LIN {X 0.009,Y -477.368,Z 1112.922,A 0.000,B 0.000,C 90.000,E1 22.025} C_DIS
LIN {X 0.039,Y -465.405,Z 1112.917,A 0.000,B 0.000,C 90.000,E1 20.972} C_DIS
LIN {X 0.095,Y -448.968,Z 1112.908,A 0.000,B 0.000,C 90.000,E1 19.504} C_DIS
LIN {X 0.026,Y -429.956,Z 1112.898,A 0.000,B 0.000,C 90.000,E1 17.692} C_DIS
LIN {X -0.246,Y -415.856,Z 1112.890,A 0.000,B 0.000,C 90.000,E1 16.205} C_DIS
LIN {X 0.123,Y -407.881,Z 1112.885,A 0.000,B 0.000,C 90.000,E1 15.190} C_DIS
LIN {X -0.086,Y -401.258,Z 1112.880,A 0.000,B 0.000,C 90.000,E1 14.356} C_DIS
LIN {X 0.152,Y -396.233,Z 1112.875,A 0.000,B 0.000,C 90.000,E1 13.536} C_DIS
LIN {X 0.076,Y -394.151,Z 1112.873,A 0.000,B 0.000,C 90.000,E1 13.119} C_DIS
LIN {X -0.071,Y -392.812,Z 1112.871,A 0.000,B 0.000,C 90.000,E1 12.703} C_DIS
LIN {X -0.136,Y -392.469,Z 1112.870,A 0.000,B 0.000,C 90.000,E1 12.535} C_DIS
LIN {X -0.161,Y -392.068,Z 1112.867,A 0.000,B 0.000,C 90.000,E1 12.007} C_DIS
LIN {X 0.211,Y -392.446,Z 1112.863,A 0.000,B 0.000,C 90.000,E1 11.243} C_DIS
LIN {X 0.042,Y -394.824,Z 1112.855,A 0.000,B 0.000,C 90.000,E1 9.849} C_DIS
LIN {X -0.112,Y -398.885,Z 1112.845,A 0.000,B 0.000,C 90.000,E1 8.106} C_DIS
LIN {X 0.165,Y -402.538,Z 1112.837,A 0.000,B 0.000,C 90.000,E1 6.663} C_DIS
LIN {X 0.148,Y -404.293,Z 1112.833,A 0.000,B 0.000,C 90.000,E1 5.967} C_DIS
LIN {X 0.101,Y -406.462,Z 1112.829,A 0.000,B 0.000,C 90.000,E1 5.277} C_DIS
LIN {X 0.083,Y -407.246,Z 1112.828,A 0.000,B 0.000,C 90.000,E1 5.106} C_DIS
LIN {X 0.015,Y -410.748,Z 1112.825,A 0.000,B 0.000,C 90.000,E1 4.531} C_DIS
LIN {X 0.005,Y -411.930,Z 1112.824,A 0.000,B 0.000,C 90.000,E1 4.359} C_DIS
LIN {X 0.157,Y -416.065,Z 1112.822,A 0.000,B 0.000,C 90.000,E1 3.955} C_DIS
LIN {X -0.197,Y -431.618,Z 1112.816,A 0.000,B 0.000,C 90.000,E1 2.922} C_DIS
LIN {X 0.226,Y -451.307,Z 1112.809,A 0.000,B 0.000,C 90.000,E1 1.547} C_DIS
LIN {X 0.037,Y -465.923,Z 1112.804,A 0.000,B 0.000,C 90.000,E1 0.630} C_DIS
LIN {X 0.181,Y -479.029,Z 1112.799,A 0.000,B 0.000,C 90.000,E1 359.771} C_DIS
LIN {X 0.170,Y -490.278,Z 1112.795,A 0.000,B 0.000,C 90.000,E1 359.026} C_DIS
LIN {X -0.165,Y -497.943,Z 1112.792,A 0.000,B 0.000,C 90.000,E1 358.511} C_DIS
LIN {X -0.165,Y -504.029,Z 1112.789,A 0.000,B 0.000,C 90.000,E1 358.051} C_DIS
LIN {X -0.251,Y -509.905,Z 1112.786,A 0.000,B 0.000,C 90.000,E1 357.593} C_DIS
LIN {X 0.073,Y -516.804,Z 1112.783,A 0.000,B 0.000,C 90.000,E1 356.963} C_DIS
LIN {X -0.071,Y -523.698,Z 1112.780,A 0.000,B 0.000,C 90.000,E1 356.331} C_DIS
LIN {X 0.049,Y -530.246,Z 1112.776,A 0.000,B 0.000,C 90.000,E1 355.641} C_DIS
LIN {X -0.178,Y -536.359,Z 1112.772,A 0.000,B 0.000,C 90.000,E1 354.951} C_DIS
LIN {X 0.132,Y -541.871,Z 1112.768,A 0.000,B 0.000,C 90.000,E1 354.204} C_DIS
LIN {X 0.212,Y -545.882,Z 1112.765,A 0.000,B 0.000,C 90.000,E1 353.628} C_DIS
LIN {X 0.129,Y -550.391,Z 1112.761,A 0.000,B 0.000,C 90.000,E1 352.932} C_DIS
LIN {X 0.274,Y -553.810,Z 1112.758,A 0.000,B 0.000,C 90.000,E1 352.356} C_DIS
LIN {X 0.269,Y -557.505,Z 1112.754,A 0.000,B 0.000,C 90.000,E1 351.659} C_DIS
LIN {X 0.210,Y -560.782,Z 1112.750,A 0.000,B 0.000,C 90.000,E1 350.971} C_DIS
LIN {X 0.112,Y -564.383,Z 1112.745,A 0.000,B 0.000,C 90.000,E1 350.151} C_DIS
LIN {X -0.050,Y -567.672,Z 1112.741,A 0.000,B 0.000,C 90.000,E1 349.342} C_DIS
LIN {X -0.075,Y -570.756,Z 1112.736,A 0.000,B 0.000,C 90.000,E1 348.522} C_DIS
LIN {X -0.065,Y -573.611,Z 1112.732,A 0.000,B 0.000,C 90.000,E1 347.701} C_DIS
LIN {X -0.025,Y -576.322,Z 1112.727,A 0.000,B 0.000,C 90.000,E1 346.881} C_DIS
LIN {X 0.039,Y -578.786,Z 1112.723,A 0.000,B 0.000,C 90.000,E1 346.061} C_DIS
LIN {X 0.154,Y -582.796,Z 1112.715,A 0.000,B 0.000,C 90.000,E1 344.700} C_DIS
LIN {X -0.131,Y -585.112,Z 1112.711,A 0.000,B 0.000,C 90.000,E1 343.921} C_DIS
LIN {X -0.065,Y -589.522,Z 1112.702,A 0.000,B 0.000,C 90.000,E1 342.308} C_DIS
LIN {X 0.024,Y -592.834,Z 1112.694,A 0.000,B 0.000,C 90.000,E1 340.967} C_DIS
LIN {X 0.287,Y -595.374,Z 1112.688,A 0.000,B 0.000,C 90.000,E1 339.880} C_DIS
LIN {X 0.329,Y -597.064,Z 1112.684,A 0.000,B 0.000,C 90.000,E1 339.082} C_DIS
LIN {X 0.079,Y -599.028,Z 1112.678,A 0.000,B 0.000,C 90.000,E1 338.050} C_DIS
LIN {X 0.070,Y -600.755,Z 1112.672,A 0.000,B 0.000,C 90.000,E1 336.997} C_DIS
LIN {X -0.154,Y -601.854,Z 1112.668,A 0.000,B 0.000,C 90.000,E1 336.230} C_DIS
LIN {X -0.127,Y -603.008,Z 1112.662,A 0.000,B 0.000,C 90.000,E1 335.177} C_DIS
LIN {X -0.319,Y -603.791,Z 1112.658,A 0.000,B 0.000,C 90.000,E1 334.409} C_DIS
LIN {X -0.019,Y -604.386,Z 1112.652,A 0.000,B 0.000,C 90.000,E1 333.332} C_DIS
LIN {X 0.081,Y -604.735,Z 1112.648,A 0.000,B 0.000,C 90.000,E1 332.538} C_DIS
LIN {X -0.208,Y -604.666,Z 1112.640,A 0.000,B 0.000,C 90.000,E1 331.257} C_DIS
LIN {X -0.156,Y -603.977,Z 1112.634,A 0.000,B 0.000,C 90.000,E1 330.205} C_DIS
LIN {X -0.049,Y -603.017,Z 1112.630,A 0.000,B 0.000,C 90.000,E1 329.410} C_DIS
LIN {X 0.121,Y -602.084,Z 1112.627,A 0.000,B 0.000,C 90.000,E1 328.869} C_DIS
LIN {X 0.206,Y -600.484,Z 1112.623,A 0.000,B 0.000,C 90.000,E1 328.074} C_DIS
LIN {X -0.235,Y -598.613,Z 1112.618,A 0.000,B 0.000,C 90.000,E1 327.327} C_DIS
LIN {X 0.132,Y -596.306,Z 1112.614,A 0.000,B 0.000,C 90.000,E1 326.501} C_DIS
LIN {X -0.016,Y -593.789,Z 1112.610,A 0.000,B 0.000,C 90.000,E1 325.722} C_DIS
LIN {X 0.300,Y -590.875,Z 1112.605,A 0.000,B 0.000,C 90.000,E1 324.895} C_DIS
LIN {X 0.103,Y -587.868,Z 1112.601,A 0.000,B 0.000,C 90.000,E1 324.116} C_DIS
LIN {X 0.154,Y -585.866,Z 1112.598,A 0.000,B 0.000,C 90.000,E1 323.577} C_DIS
LIN {X 0.067,Y -583.672,Z 1112.595,A 0.000,B 0.000,C 90.000,E1 323.050} C_DIS
LIN {X -0.032,Y -579.142,Z 1112.589,A 0.000,B 0.000,C 90.000,E1 321.984} C_DIS
LIN {X -0.155,Y -576.744,Z 1112.586,A 0.000,B 0.000,C 90.000,E1 321.457} C_DIS
LIN {X 0.044,Y -573.482,Z 1112.582,A 0.000,B 0.000,C 90.000,E1 320.759} C_DIS
LIN {X 0.067,Y -568.213,Z 1112.576,A 0.000,B 0.000,C 90.000,E1 319.666} C_DIS
LIN {X -0.255,Y -564.630,Z 1112.572,A 0.000,B 0.000,C 90.000,E1 319.013} C_DIS
LIN {X -0.102,Y -561.501,Z 1112.569,A 0.000,B 0.000,C 90.000,E1 318.447} C_DIS
LIN {X 0.074,Y -558.208,Z 1112.566,A 0.000,B 0.000,C 90.000,E1 317.877} C_DIS
LIN {X 0.183,Y -554.625,Z 1112.563,A 0.000,B 0.000,C 90.000,E1 317.310} C_DIS
LIN {X -0.049,Y -546.654,Z 1112.557,A 0.000,B 0.000,C 90.000,E1 316.215} C_DIS
LIN {X -0.215,Y -543.688,Z 1112.554,A 0.000,B 0.000,C 90.000,E1 315.810} C_DIS
LIN {X -0.008,Y -540.915,Z 1112.552,A 0.000,B 0.000,C 90.000,E1 315.364} C_DIS
LIN {X -0.214,Y -537.011,Z 1112.548,A 0.000,B 0.000,C 90.000,E1 314.676} C_DIS
LIN {X 0.330,Y -535.070,Z 1112.546,A 0.000,B 0.000,C 90.000,E1 314.190} C_DIS
LIN {X 0.005,Y -533.099,Z 1112.543,A 0.000,B 0.000,C 90.000,E1 313.662} C_DIS
LIN {X 0.029,Y -531.114,Z 1112.538,A 0.000,B 0.000,C 90.000,E1 312.894} C_DIS
LIN {X 0.003,Y -530.609,Z 1112.537,A 0.000,B 0.000,C 90.000,E1 312.609} C_DIS
LIN {X -0.084,Y -529.964,Z 1112.534,A 0.000,B 0.000,C 90.000,E1 312.043} C_DIS
LIN {X -0.111,Y -529.478,Z 1112.532,A 0.000,B 0.000,C 90.000,E1 311.757} C_DIS
LIN {X -0.136,Y -529.401,Z 1112.530,A 0.000,B 0.000,C 90.000,E1 311.472} C_DIS
LIN {X 0.162,Y -528.898,Z 1112.527,A 0.000,B 0.000,C 90.000,E1 310.862} C_DIS
LIN {X 0.052,Y -528.782,Z 1112.524,A 0.000,B 0.000,C 90.000,E1 310.297} C_DIS
LIN {X 0.290,Y -528.759,Z 1112.518,A 0.000,B 0.000,C 90.000,E1 309.116} C_DIS
LIN {X 0.096,Y -529.954,Z 1112.501,A 0.000,B 0.000,C 90.000,E1 306.251} C_DIS
LIN {X -0.018,Y -531.286,Z 1112.490,A 0.000,B 0.000,C 90.000,E1 304.246} C_DIS
LIN {X -0.260,Y -532.419,Z 1112.481,A 0.000,B 0.000,C 90.000,E1 302.546} C_DIS
LIN {X -0.019,Y -533.825,Z 1112.471,A 0.000,B 0.000,C 90.000,E1 300.797} C_DIS
LIN {X -0.020,Y -535.088,Z 1112.462,A 0.000,B 0.000,C 90.000,E1 299.077} C_DIS
LIN {X -0.141,Y -535.607,Z 1112.457,A 0.000,B 0.000,C 90.000,E1 298.231} C_DIS
LIN {X -0.092,Y -536.415,Z 1112.449,A 0.000,B 0.000,C 90.000,E1 296.796} C_DIS
LIN {X 0.038,Y -536.763,Z 1112.444,A 0.000,B 0.000,C 90.000,E1 295.924} C_DIS
LIN {X -0.139,Y -537.151,Z 1112.436,A 0.000,B 0.000,C 90.000,E1 294.515} C_DIS
LIN {X -0.051,Y -537.438,Z 1112.428,A 0.000,B 0.000,C 90.000,E1 293.078} C_DIS
LIN {X -0.161,Y -537.544,Z 1112.420,A 0.000,B 0.000,C 90.000,E1 291.663} C_DIS
LIN {X -0.266,Y -537.534,Z 1112.412,A 0.000,B 0.000,C 90.000,E1 290.248} C_DIS
LIN {X -0.089,Y -537.427,Z 1112.406,A 0.000,B 0.000,C 90.000,E1 289.087} C_DIS
LIN {X -0.139,Y -536.979,Z 1112.395,A 0.000,B 0.000,C 90.000,E1 287.094} C_DIS
LIN {X -0.046,Y -536.434,Z 1112.385,A 0.000,B 0.000,C 90.000,E1 285.371} C_DIS
LIN {X -0.207,Y -535.915,Z 1112.379,A 0.000,B 0.000,C 90.000,E1 284.245} C_DIS
LIN {X -0.214,Y -534.929,Z 1112.368,A 0.000,B 0.000,C 90.000,E1 282.243} C_DIS
LIN {X 0.058,Y -534.206,Z 1112.360,A 0.000,B 0.000,C 90.000,E1 280.782} C_DIS
LIN {X -0.170,Y -533.353,Z 1112.350,A 0.000,B 0.000,C 90.000,E1 279.086} C_DIS
LIN {X -0.096,Y -532.371,Z 1112.339,A 0.000,B 0.000,C 90.000,E1 277.068} C_DIS
LIN {X -0.039,Y -531.638,Z 1112.331,A 0.000,B 0.000,C 90.000,E1 275.625} C_DIS
LIN {X -0.051,Y -530.744,Z 1112.320,A 0.000,B 0.000,C 90.000,E1 273.612} C_DIS
LIN {X -0.111,Y -530.074,Z 1112.312,A 0.000,B 0.000,C 90.000,E1 272.178} C_DIS
LIN {X -0.203,Y -529.294,Z 1112.302,A 0.000,B 0.000,C 90.000,E1 270.458} C_DIS
LIN {X -0.262,Y -528.907,Z 1112.298,A 0.000,B 0.000,C 90.000,E1 269.599} C_DIS
LIN {X 0.149,Y -528.050,Z 1112.288,A 0.000,B 0.000,C 90.000,E1 267.822} C_DIS
LIN {X 0.038,Y -527.174,Z 1112.280,A 0.000,B 0.000,C 90.000,E1 266.388} C_DIS
LIN {X -0.096,Y -526.057,Z 1112.270,A 0.000,B 0.000,C 90.000,E1 264.666} C_DIS
LIN {X -0.173,Y -525.177,Z 1112.264,A 0.000,B 0.000,C 90.000,E1 263.514} C_DIS
LIN {X -0.197,Y -524.077,Z 1112.257,A 0.000,B 0.000,C 90.000,E1 262.356} C_DIS
LIN {X 0.232,Y -521.513,Z 1112.243,A 0.000,B 0.000,C 90.000,E1 259.690} C_DIS
LIN {X 0.247,Y -519.858,Z 1112.233,A 0.000,B 0.000,C 90.000,E1 257.937} C_DIS
LIN {X -0.175,Y -517.933,Z 1112.222,A 0.000,B 0.000,C 90.000,E1 255.936} C_DIS
LIN {X -0.100,Y -516.792,Z 1112.215,A 0.000,B 0.000,C 90.000,E1 254.755} C_DIS
LIN {X 0.095,Y -515.517,Z 1112.209,A 0.000,B 0.000,C 90.000,E1 253.559} C_DIS
LIN {X -0.136,Y -513.723,Z 1112.199,A 0.000,B 0.000,C 90.000,E1 251.819} C_DIS
LIN {X 0.120,Y -512.149,Z 1112.191,A 0.000,B 0.000,C 90.000,E1 250.315} C_DIS
LIN {X 0.139,Y -510.097,Z 1112.181,A 0.000,B 0.000,C 90.000,E1 248.539} C_DIS
LIN {X -0.166,Y -507.911,Z 1112.171,A 0.000,B 0.000,C 90.000,E1 246.794} C_DIS
LIN {X 0.129,Y -506.655,Z 1112.166,A 0.000,B 0.000,C 90.000,E1 245.869} C_DIS
LIN {X -0.216,Y -504.978,Z 1112.159,A 0.000,B 0.000,C 90.000,E1 244.717} C_DIS
LIN {X -0.124,Y -503.108,Z 1112.153,A 0.000,B 0.000,C 90.000,E1 243.512} C_DIS
LIN {X 0.077,Y -500.227,Z 1112.143,A 0.000,B 0.000,C 90.000,E1 241.691} C_DIS
LIN {X 0.031,Y -498.747,Z 1112.138,A 0.000,B 0.000,C 90.000,E1 240.795} C_DIS
LIN {X -0.059,Y -495.801,Z 1112.128,A 0.000,B 0.000,C 90.000,E1 238.997} C_DIS
LIN {X -0.069,Y -493.686,Z 1112.121,A 0.000,B 0.000,C 90.000,E1 237.788} C_DIS
LIN {X -0.020,Y -490.521,Z 1112.111,A 0.000,B 0.000,C 90.000,E1 235.960} C_DIS
LIN {X 0.264,Y -487.817,Z 1112.102,A 0.000,B 0.000,C 90.000,E1 234.402} C_DIS
LIN {X -0.179,Y -484.923,Z 1112.094,A 0.000,B 0.000,C 90.000,E1 232.924} C_DIS
LIN {X 0.104,Y -481.406,Z 1112.084,A 0.000,B 0.000,C 90.000,E1 231.045} C_DIS
LIN {X -0.048,Y -479.034,Z 1112.077,A 0.000,B 0.000,C 90.000,E1 229.828} C_DIS
LIN {X 0.237,Y -476.005,Z 1112.068,A 0.000,B 0.000,C 90.000,E1 228.243} C_DIS
LIN {X 0.200,Y -472.520,Z 1112.058,A 0.000,B 0.000,C 90.000,E1 226.377} C_DIS
LIN {X 0.070,Y -469.061,Z 1112.047,A 0.000,B 0.000,C 90.000,E1 224.514} C_DIS
LIN {X 0.130,Y -466.300,Z 1112.039,A 0.000,B 0.000,C 90.000,E1 222.933} C_DIS
LIN {X -0.121,Y -463.116,Z 1112.028,A 0.000,B 0.000,C 90.000,E1 221.067} C_DIS
LIN {X -0.012,Y -459.634,Z 1112.016,A 0.000,B 0.000,C 90.000,E1 218.830} C_DIS
LIN {X 0.075,Y -456.279,Z 1112.003,A 0.000,B 0.000,C 90.000,E1 216.583} C_DIS
LIN {X 0.090,Y -454.065,Z 1111.994,A 0.000,B 0.000,C 90.000,E1 214.978} C_DIS
LIN {X 0.063,Y -451.814,Z 1111.985,A 0.000,B 0.000,C 90.000,E1 213.372} C_DIS
LIN {X -0.099,Y -448.884,Z 1111.973,A 0.000,B 0.000,C 90.000,E1 211.131} C_DIS
LIN {X 0.198,Y -446.213,Z 1111.960,A 0.000,B 0.000,C 90.000,E1 208.821} C_DIS
LIN {X 0.006,Y -444.131,Z 1111.948,A 0.000,B 0.000,C 90.000,E1 206.565} C_DIS
LIN {X 0.114,Y -443.057,Z 1111.937,A 0.000,B 0.000,C 90.000,E1 204.591} C_DIS
LIN {X 0.156,Y -443.425,Z 1111.928,A 0.000,B 0.000,C 90.000,E1 202.950} C_DIS
LIN {X 0.002,Y -444.595,Z 1111.920,A 0.000,B 0.000,C 90.000,E1 201.663} C_DIS
LIN {X -0.114,Y -445.583,Z 1111.917,A 0.000,B 0.000,C 90.000,E1 201.025} C_DIS
LIN {X -0.259,Y -447.580,Z 1111.911,A 0.000,B 0.000,C 90.000,E1 200.066} C_DIS
LIN {X -0.044,Y -451.809,Z 1111.902,A 0.000,B 0.000,C 90.000,E1 198.417} C_DIS
LIN {X 0.073,Y -459.189,Z 1111.890,A 0.000,B 0.000,C 90.000,E1 196.150} C_DIS
LIN {X 0.227,Y -470.714,Z 1111.873,A 0.000,B 0.000,C 90.000,E1 193.119} C_DIS
LIN {X 0.094,Y -479.895,Z 1111.861,A 0.000,B 0.000,C 90.000,E1 190.950} C_DIS
LIN {X -0.116,Y -488.663,Z 1111.850,A 0.000,B 0.000,C 90.000,E1 188.973} C_DIS
LIN {X -0.095,Y -496.045,Z 1111.841,A 0.000,B 0.000,C 90.000,E1 187.296} C_DIS
LIN {X -0.165,Y -502.571,Z 1111.832,A 0.000,B 0.000,C 90.000,E1 185.796} C_DIS
LIN {X 0.188,Y -511.586,Z 1111.821,A 0.000,B 0.000,C 90.000,E1 183.669} C_DIS
LIN {X 0.112,Y -517.370,Z 1111.813,A 0.000,B 0.000,C 90.000,E1 182.350} C_DIS
LIN {X 0.047,Y -525.847,Z 1111.803,A 0.000,B 0.000,C 90.000,E1 180.458} C_DIS
LIN {X 0.182,Y -532.968,Z 1111.794,A 0.000,B 0.000,C 90.000,E1 178.854} C_DIS
LIN {X -0.065,Y -540.073,Z 1111.785,A 0.000,B 0.000,C 90.000,E1 177.306} C_DIS
LIN {X 0.112,Y -546.498,Z 1111.777,A 0.000,B 0.000,C 90.000,E1 175.869} C_DIS
LIN {X 0.064,Y -552.222,Z 1111.770,A 0.000,B 0.000,C 90.000,E1 174.609} C_DIS
LIN {X -0.145,Y -560.503,Z 1111.760,A 0.000,B 0.000,C 90.000,E1 172.818} C_DIS
LIN {X -0.095,Y -566.810,Z 1111.752,A 0.000,B 0.000,C 90.000,E1 171.432} C_DIS
LIN {X -0.085,Y -573.537,Z 1111.744,A 0.000,B 0.000,C 90.000,E1 169.926} C_DIS
LIN {X -0.182,Y -579.558,Z 1111.736,A 0.000,B 0.000,C 90.000,E1 168.578} C_DIS
LIN {X 0.158,Y -584.140,Z 1111.730,A 0.000,B 0.000,C 90.000,E1 167.465} C_DIS
LIN {X -0.259,Y -587.510,Z 1111.726,A 0.000,B 0.000,C 90.000,E1 166.700} C_DIS
LIN {X 0.184,Y -591.788,Z 1111.720,A 0.000,B 0.000,C 90.000,E1 165.589} C_DIS
LIN {X -0.013,Y -594.883,Z 1111.716,A 0.000,B 0.000,C 90.000,E1 164.810} C_DIS
LIN {X -0.183,Y -599.654,Z 1111.708,A 0.000,B 0.000,C 90.000,E1 163.504} C_DIS
LIN {X -0.296,Y -602.396,Z 1111.704,A 0.000,B 0.000,C 90.000,E1 162.725} C_DIS
LIN {X -0.170,Y -606.635,Z 1111.697,A 0.000,B 0.000,C 90.000,E1 161.402} C_DIS
LIN {X -0.286,Y -609.858,Z 1111.691,A 0.000,B 0.000,C 90.000,E1 160.369} C_DIS
LIN {X -0.144,Y -612.911,Z 1111.685,A 0.000,B 0.000,C 90.000,E1 159.316} C_DIS
LIN {X -0.174,Y -615.788,Z 1111.679,A 0.000,B 0.000,C 90.000,E1 158.284} C_DIS
LIN {X -0.219,Y -619.981,Z 1111.671,A 0.000,B 0.000,C 90.000,E1 156.741} C_DIS
LIN {X 0.057,Y -623.295,Z 1111.664,A 0.000,B 0.000,C 90.000,E1 155.433} C_DIS
LIN {X 0.076,Y -625.894,Z 1111.658,A 0.000,B 0.000,C 90.000,E1 154.409} C_DIS
LIN {X 0.157,Y -628.951,Z 1111.651,A 0.000,B 0.000,C 90.000,E1 153.127} C_DIS
LIN {X -0.271,Y -631.792,Z 1111.644,A 0.000,B 0.000,C 90.000,E1 151.897} C_DIS
LIN {X 0.205,Y -634.592,Z 1111.637,A 0.000,B 0.000,C 90.000,E1 150.589} C_DIS
LIN {X 0.220,Y -637.771,Z 1111.628,A 0.000,B 0.000,C 90.000,E1 149.076} C_DIS
LIN {X -0.309,Y -640.299,Z 1111.621,A 0.000,B 0.000,C 90.000,E1 147.867} C_DIS
LIN {X 0.081,Y -642.717,Z 1111.614,A 0.000,B 0.000,C 90.000,E1 146.580} C_DIS
LIN {X -0.076,Y -644.570,Z 1111.609,A 0.000,B 0.000,C 90.000,E1 145.595} C_DIS
LIN {X -0.156,Y -646.753,Z 1111.602,A 0.000,B 0.000,C 90.000,E1 144.356} C_DIS
LIN {X 0.084,Y -649.389,Z 1111.594,A 0.000,B 0.000,C 90.000,E1 142.844} C_DIS
LIN {X -0.156,Y -652.964,Z 1111.583,A 0.000,B 0.000,C 90.000,E1 140.884} C_DIS
LIN {X -0.400,Y -656.643,Z 1111.572,A 0.000,B 0.000,C 90.000,E1 138.933} C_DIS
LIN {X 0.354,Y -660.001,Z 1111.562,A 0.000,B 0.000,C 90.000,E1 137.148} C_DIS
LIN {X -0.236,Y -664.132,Z 1111.551,A 0.000,B 0.000,C 90.000,E1 135.243} C_DIS
LIN {X 0.230,Y -669.230,Z 1111.539,A 0.000,B 0.000,C 90.000,E1 133.014} C_DIS
LIN {X -0.060,Y -674.540,Z 1111.527,A 0.000,B 0.000,C 90.000,E1 130.862} C_DIS
LIN {X 0.138,Y -678.079,Z 1111.519,A 0.000,B 0.000,C 90.000,E1 129.402} C_DIS
LIN {X 0.070,Y -681.801,Z 1111.511,A 0.000,B 0.000,C 90.000,E1 127.971} C_DIS
LIN {X 0.088,Y -685.476,Z 1111.503,A 0.000,B 0.000,C 90.000,E1 126.537} C_DIS
LIN {X 0.325,Y -687.268,Z 1111.499,A 0.000,B 0.000,C 90.000,E1 125.804} C_DIS
LIN {X -0.325,Y -691.332,Z 1111.490,A 0.000,B 0.000,C 90.000,E1 124.199} C_DIS
LIN {X 0.036,Y -694.817,Z 1111.482,A 0.000,B 0.000,C 90.000,E1 122.752} C_DIS
LIN {X 0.185,Y -697.012,Z 1111.477,A 0.000,B 0.000,C 90.000,E1 121.799} C_DIS
LIN {X -0.257,Y -698.517,Z 1111.473,A 0.000,B 0.000,C 90.000,E1 121.131} C_DIS
LIN {X -0.082,Y -699.870,Z 1111.469,A 0.000,B 0.000,C 90.000,E1 120.413} C_DIS
LIN {X 0.119,Y -701.498,Z 1111.464,A 0.000,B 0.000,C 90.000,E1 119.461} C_DIS
LIN {X -0.015,Y -702.954,Z 1111.459,A 0.000,B 0.000,C 90.000,E1 118.537} C_DIS
LIN {X 0.158,Y -704.253,Z 1111.453,A 0.000,B 0.000,C 90.000,E1 117.590} C_DIS
LIN {X -0.236,Y -704.918,Z 1111.449,A 0.000,B 0.000,C 90.000,E1 116.924} C_DIS
LIN {X 0.262,Y -705.762,Z 1111.443,A 0.000,B 0.000,C 90.000,E1 115.720} C_DIS
LIN {X 0.195,Y -705.963,Z 1111.439,A 0.000,B 0.000,C 90.000,E1 115.027} C_DIS
LIN {X -0.158,Y -705.902,Z 1111.437,A 0.000,B 0.000,C 90.000,E1 114.591} C_DIS
LIN {X -0.221,Y -705.136,Z 1111.434,A 0.000,B 0.000,C 90.000,E1 114.131} C_DIS
LIN {X -0.220,Y -704.594,Z 1111.433,A 0.000,B 0.000,C 90.000,E1 113.898} C_DIS
LIN {X 0.348,Y -702.685,Z 1111.430,A 0.000,B 0.000,C 90.000,E1 113.387} C_DIS
LIN {X -0.436,Y -702.113,Z 1111.429,A 0.000,B 0.000,C 90.000,E1 113.334} C_DIS
LIN {X -0.297,Y -701.240,Z 1111.429,A 0.000,B 0.000,C 90.000,E1 113.206} C_DIS
LIN {X -0.029,Y -696.964,Z 1111.426,A 0.000,B 0.000,C 90.000,E1 112.717} C_DIS
LIN {X 0.099,Y -695.384,Z 1111.426,A 0.000,B 0.000,C 90.000,E1 112.589} C_DIS
LIN {X -0.014,Y -690.978,Z 1111.425,A 0.000,B 0.000,C 90.000,E1 112.408} C_DIS
LIN {X -0.072,Y -685.718,Z 1111.423,A 0.000,B 0.000,C 90.000,E1 112.206} C_DIS
LIN {X 0.066,Y -683.449,Z 1111.423,A 0.000,B 0.000,C 90.000,E1 112.153} C_DIS
LIN {X 0.059,Y -676.047,Z 1111.423,A 0.000,B 0.000,C 90.000,E1 112.078} C_DIS
LIN {X 0.013,Y -603.763,Z 1111.423,A 0.000,B 0.000,C 90.000,E1 112.078} C_DIS
LIN {X 0.029,Y -600.557,Z 1111.422,A 0.000,B 0.000,C 90.000,E1 111.897} C_DIS
LIN {X 0.111,Y -594.792,Z 1111.419,A 0.000,B 0.000,C 90.000,E1 111.461} C_DIS
LIN {X 0.166,Y -587.133,Z 1111.416,A 0.000,B 0.000,C 90.000,E1 110.791} C_DIS
LIN {X 0.151,Y -578.854,Z 1111.412,A 0.000,B 0.000,C 90.000,E1 110.066} C_DIS
LIN {X 0.192,Y -574.638,Z 1111.410,A 0.000,B 0.000,C 90.000,E1 109.704} C_DIS
LIN {X -0.003,Y -568.549,Z 1111.407,A 0.000,B 0.000,C 90.000,E1 109.268} C_DIS
LIN {X 0.255,Y -560.311,Z 1111.404,A 0.000,B 0.000,C 90.000,E1 108.725} C_DIS
LIN {X 0.085,Y -553.963,Z 1111.402,A 0.000,B 0.000,C 90.000,E1 108.362} C_DIS
LIN {X -0.188,Y -550.006,Z 1111.401,A 0.000,B 0.000,C 90.000,E1 108.109} C_DIS
LIN {X 0.258,Y -548.776,Z 1111.400,A 0.000,B 0.000,C 90.000,E1 107.873} C_DIS
LIN {X 0.216,Y -548.757,Z 1111.399,A 0.000,B 0.000,C 90.000,E1 107.873} C_DIS
LIN {X -0.099,Y -548.411,Z 1111.397,A 0.000,B 0.000,C 90.000,E1 107.511} C_DIS
LIN {X 0.075,Y -548.753,Z 1111.393,A 0.000,B 0.000,C 90.000,E1 106.732} C_DIS
LIN {X 0.084,Y -549.554,Z 1111.387,A 0.000,B 0.000,C 90.000,E1 105.607} C_DIS
LIN {X 0.261,Y -551.471,Z 1111.373,A 0.000,B 0.000,C 90.000,E1 103.063} C_DIS
LIN {X 0.009,Y -553.177,Z 1111.362,A 0.000,B 0.000,C 90.000,E1 101.130} C_DIS
LIN {X 0.114,Y -554.811,Z 1111.353,A 0.000,B 0.000,C 90.000,E1 99.443} C_DIS
LIN {X 0.250,Y -556.528,Z 1111.343,A 0.000,B 0.000,C 90.000,E1 97.757} C_DIS
LIN {X -0.158,Y -558.492,Z 1111.333,A 0.000,B 0.000,C 90.000,E1 95.853} C_DIS
LIN {X -0.230,Y -559.689,Z 1111.325,A 0.000,B 0.000,C 90.000,E1 94.473} C_DIS
LIN {X 0.274,Y -560.766,Z 1111.317,A 0.000,B 0.000,C 90.000,E1 93.037} C_DIS
LIN {X 0.089,Y -561.446,Z 1111.311,A 0.000,B 0.000,C 90.000,E1 91.949} C_DIS
LIN {X 0.035,Y -562.276,Z 1111.303,A 0.000,B 0.000,C 90.000,E1 90.573} C_DIS
LIN {X -0.018,Y -562.972,Z 1111.296,A 0.000,B 0.000,C 90.000,E1 89.198} C_DIS
LIN {X 0.058,Y -563.839,Z 1111.286,A 0.000,B 0.000,C 90.000,E1 87.535} C_DIS
LIN {X 0.185,Y -564.611,Z 1111.277,A 0.000,B 0.000,C 90.000,E1 85.869} C_DIS
LIN {X -0.082,Y -565.364,Z 1111.266,A 0.000,B 0.000,C 90.000,E1 83.970} C_DIS
LIN {X 0.290,Y -566.130,Z 1111.256,A 0.000,B 0.000,C 90.000,E1 82.008} C_DIS
LIN {X 0.191,Y -566.832,Z 1111.245,A 0.000,B 0.000,C 90.000,E1 80.095} C_DIS
LIN {X 0.022,Y -567.505,Z 1111.236,A 0.000,B 0.000,C 90.000,E1 78.465} C_DIS
LIN {X -0.026,Y -568.295,Z 1111.227,A 0.000,B 0.000,C 90.000,E1 76.825} C_DIS
LIN {X 0.199,Y -569.676,Z 1111.213,A 0.000,B 0.000,C 90.000,E1 74.338} C_DIS
LIN {X -0.097,Y -571.244,Z 1111.201,A 0.000,B 0.000,C 90.000,E1 72.181} C_DIS
LIN {X 0.182,Y -573.217,Z 1111.187,A 0.000,B 0.000,C 90.000,E1 69.699} C_DIS
LIN {X 0.192,Y -574.425,Z 1111.180,A 0.000,B 0.000,C 90.000,E1 68.337} C_DIS
LIN {X 0.231,Y -575.716,Z 1111.172,A 0.000,B 0.000,C 90.000,E1 66.975} C_DIS
LIN {X -0.018,Y -577.324,Z 1111.162,A 0.000,B 0.000,C 90.000,E1 65.101} C_DIS
LIN {X -0.230,Y -578.399,Z 1111.154,A 0.000,B 0.000,C 90.000,E1 63.768} C_DIS
LIN {X 0.208,Y -579.564,Z 1111.145,A 0.000,B 0.000,C 90.000,E1 62.103} C_DIS
LIN {X -0.216,Y -580.819,Z 1111.135,A 0.000,B 0.000,C 90.000,E1 60.255} C_DIS
LIN {X 0.172,Y -581.619,Z 1111.127,A 0.000,B 0.000,C 90.000,E1 58.869} C_DIS
LIN {X 0.212,Y -582.297,Z 1111.121,A 0.000,B 0.000,C 90.000,E1 57.788} C_DIS
LIN {X -0.026,Y -583.232,Z 1111.111,A 0.000,B 0.000,C 90.000,E1 55.928} C_DIS
LIN {X -0.090,Y -584.056,Z 1111.102,A 0.000,B 0.000,C 90.000,E1 54.322} C_DIS
LIN {X -0.245,Y -584.944,Z 1111.090,A 0.000,B 0.000,C 90.000,E1 52.190} C_DIS
LIN {X 0.040,Y -585.158,Z 1111.084,A 0.000,B 0.000,C 90.000,E1 51.090} C_DIS
LIN {X 0.144,Y -585.281,Z 1111.079,A 0.000,B 0.000,C 90.000,E1 50.275} C_DIS
LIN {X 0.165,Y -585.200,Z 1111.072,A 0.000,B 0.000,C 90.000,E1 48.933} C_DIS
LIN {X -0.002,Y -585.032,Z 1111.066,A 0.000,B 0.000,C 90.000,E1 47.877} C_DIS
LIN {X 0.218,Y -584.729,Z 1111.060,A 0.000,B 0.000,C 90.000,E1 46.782} C_DIS
LIN {X -0.245,Y -584.197,Z 1111.053,A 0.000,B 0.000,C 90.000,E1 45.486} C_DIS
LIN {X -0.044,Y -583.562,Z 1111.047,A 0.000,B 0.000,C 90.000,E1 44.393} C_DIS
LIN {X 0.012,Y -582.954,Z 1111.042,A 0.000,B 0.000,C 90.000,E1 43.581} C_DIS
LIN {X -0.217,Y -581.967,Z 1111.036,A 0.000,B 0.000,C 90.000,E1 42.528} C_DIS
LIN {X 0.068,Y -581.311,Z 1111.033,A 0.000,B 0.000,C 90.000,E1 41.962} C_DIS
LIN {X -0.156,Y -579.979,Z 1111.027,A 0.000,B 0.000,C 90.000,E1 40.906} C_DIS
LIN {X -0.112,Y -578.921,Z 1111.023,A 0.000,B 0.000,C 90.000,E1 40.092} C_DIS
LIN {X -0.208,Y -576.639,Z 1111.015,A 0.000,B 0.000,C 90.000,E1 38.749} C_DIS
LIN {X 0.254,Y -575.062,Z 1111.011,A 0.000,B 0.000,C 90.000,E1 37.890} C_DIS
LIN {X 0.245,Y -573.236,Z 1111.006,A 0.000,B 0.000,C 90.000,E1 37.076} C_DIS
LIN {X -0.129,Y -571.225,Z 1111.002,A 0.000,B 0.000,C 90.000,E1 36.297} C_DIS
LIN {X 0.008,Y -570.520,Z 1111.000,A 0.000,B 0.000,C 90.000,E1 36.011} C_DIS
LIN {X 0.070,Y -567.941,Z 1110.996,A 0.000,B 0.000,C 90.000,E1 35.185} C_DIS
LIN {X -0.354,Y -565.171,Z 1110.991,A 0.000,B 0.000,C 90.000,E1 34.405} C_DIS
LIN {X -0.242,Y -564.159,Z 1110.990,A 0.000,B 0.000,C 90.000,E1 34.119} C_DIS
LIN {X -0.242,Y -560.733,Z 1110.985,A 0.000,B 0.000,C 90.000,E1 33.293} C_DIS
LIN {X 0.191,Y -557.057,Z 1110.980,A 0.000,B 0.000,C 90.000,E1 32.418} C_DIS
LIN {X 0.104,Y -552.952,Z 1110.976,A 0.000,B 0.000,C 90.000,E1 31.592} C_DIS
LIN {X -0.196,Y -549.302,Z 1110.972,A 0.000,B 0.000,C 90.000,E1 30.924} C_DIS
LIN {X -0.176,Y -544.633,Z 1110.967,A 0.000,B 0.000,C 90.000,E1 30.079} C_DIS
LIN {X 0.196,Y -540.523,Z 1110.963,A 0.000,B 0.000,C 90.000,E1 29.333} C_DIS
LIN {X -0.335,Y -536.954,Z 1110.960,A 0.000,B 0.000,C 90.000,E1 28.821} C_DIS
LIN {X -0.158,Y -533.062,Z 1110.957,A 0.000,B 0.000,C 90.000,E1 28.231} C_DIS
LIN {X -0.161,Y -527.800,Z 1110.953,A 0.000,B 0.000,C 90.000,E1 27.513} C_DIS
LIN {X -0.058,Y -523.395,Z 1110.950,A 0.000,B 0.000,C 90.000,E1 26.924} C_DIS
LIN {X -0.062,Y -519.909,Z 1110.947,A 0.000,B 0.000,C 90.000,E1 26.488} C_DIS
LIN {X 0.292,Y -513.604,Z 1110.943,A 0.000,B 0.000,C 90.000,E1 25.720} C_DIS
LIN {X -0.129,Y -505.696,Z 1110.938,A 0.000,B 0.000,C 90.000,E1 24.899} C_DIS
LIN {X -0.083,Y -496.065,Z 1110.933,A 0.000,B 0.000,C 90.000,E1 23.898} C_DIS
LIN {X -0.165,Y -486.110,Z 1110.927,A 0.000,B 0.000,C 90.000,E1 22.950} C_DIS
LIN {X -0.178,Y -477.456,Z 1110.923,A 0.000,B 0.000,C 90.000,E1 22.153} C_DIS
LIN {X 0.185,Y -470.038,Z 1110.919,A 0.000,B 0.000,C 90.000,E1 21.461} C_DIS
LIN {X -0.138,Y -457.051,Z 1110.913,A 0.000,B 0.000,C 90.000,E1 20.355} C_DIS
LIN {X 0.015,Y -435.079,Z 1110.902,A 0.000,B 0.000,C 90.000,E1 18.308} C_DIS
LIN {X 0.093,Y -422.326,Z 1110.895,A 0.000,B 0.000,C 90.000,E1 16.985} C_DIS
LIN {X -0.219,Y -411.437,Z 1110.888,A 0.000,B 0.000,C 90.000,E1 15.788} C_DIS
LIN {X 0.025,Y -401.084,Z 1110.880,A 0.000,B 0.000,C 90.000,E1 14.426} C_DIS
LIN {X 0.078,Y -396.147,Z 1110.876,A 0.000,B 0.000,C 90.000,E1 13.647} C_DIS
LIN {X 0.048,Y -394.506,Z 1110.874,A 0.000,B 0.000,C 90.000,E1 13.300} C_DIS
LIN {X 0.074,Y -393.770,Z 1110.873,A 0.000,B 0.000,C 90.000,E1 13.119} C_DIS
LIN {X -0.137,Y -392.324,Z 1110.870,A 0.000,B 0.000,C 90.000,E1 12.591} C_DIS
LIN {X 0.138,Y -391.973,Z 1110.867,A 0.000,B 0.000,C 90.000,E1 12.007} C_DIS
LIN {X -0.119,Y -392.534,Z 1110.863,A 0.000,B 0.000,C 90.000,E1 11.299} C_DIS
LIN {X 0.063,Y -395.659,Z 1110.853,A 0.000,B 0.000,C 90.000,E1 9.500} C_DIS
LIN {X -0.053,Y -398.954,Z 1110.845,A 0.000,B 0.000,C 90.000,E1 8.106} C_DIS
LIN {X -0.173,Y -402.562,Z 1110.837,A 0.000,B 0.000,C 90.000,E1 6.720} C_DIS
LIN {X 0.210,Y -404.272,Z 1110.833,A 0.000,B 0.000,C 90.000,E1 5.967} C_DIS
LIN {X 0.163,Y -406.373,Z 1110.829,A 0.000,B 0.000,C 90.000,E1 5.277} C_DIS
LIN {X 0.146,Y -407.055,Z 1110.828,A 0.000,B 0.000,C 90.000,E1 5.106} C_DIS
LIN {X -0.132,Y -410.515,Z 1110.825,A 0.000,B 0.000,C 90.000,E1 4.531} C_DIS
LIN {X -0.144,Y -411.729,Z 1110.824,A 0.000,B 0.000,C 90.000,E1 4.359} C_DIS
LIN {X 0.000,Y -415.683,Z 1110.822,A 0.000,B 0.000,C 90.000,E1 3.955} C_DIS
LIN {X 0.208,Y -417.440,Z 1110.821,A 0.000,B 0.000,C 90.000,E1 3.784} C_DIS
LIN {X -0.031,Y -426.335,Z 1110.818,A 0.000,B 0.000,C 90.000,E1 3.212} C_DIS
LIN {X -0.183,Y -446.085,Z 1110.810,A 0.000,B 0.000,C 90.000,E1 1.892} C_DIS
LIN {X -0.185,Y -465.636,Z 1110.803,A 0.000,B 0.000,C 90.000,E1 0.630} C_DIS
LIN {X 0.181,Y -478.333,Z 1110.799,A 0.000,B 0.000,C 90.000,E1 359.771} C_DIS
LIN {X 0.122,Y -488.018,Z 1110.795,A 0.000,B 0.000,C 90.000,E1 359.141} C_DIS
LIN {X -0.161,Y -495.830,Z 1110.792,A 0.000,B 0.000,C 90.000,E1 358.625} C_DIS
LIN {X -0.118,Y -503.463,Z 1110.789,A 0.000,B 0.000,C 90.000,E1 358.051} C_DIS
LIN {X -0.235,Y -509.453,Z 1110.786,A 0.000,B 0.000,C 90.000,E1 357.593} C_DIS
LIN {X -0.022,Y -516.607,Z 1110.783,A 0.000,B 0.000,C 90.000,E1 356.963} C_DIS
LIN {X -0.148,Y -523.521,Z 1110.780,A 0.000,B 0.000,C 90.000,E1 356.331} C_DIS
LIN {X 0.016,Y -530.077,Z 1110.776,A 0.000,B 0.000,C 90.000,E1 355.641} C_DIS
LIN {X -0.173,Y -536.221,Z 1110.772,A 0.000,B 0.000,C 90.000,E1 354.951} C_DIS
LIN {X 0.136,Y -541.768,Z 1110.768,A 0.000,B 0.000,C 90.000,E1 354.204} C_DIS
LIN {X 0.216,Y -545.879,Z 1110.765,A 0.000,B 0.000,C 90.000,E1 353.628} C_DIS
LIN {X 0.133,Y -550.441,Z 1110.761,A 0.000,B 0.000,C 90.000,E1 352.932} C_DIS
LIN {X 0.277,Y -553.872,Z 1110.758,A 0.000,B 0.000,C 90.000,E1 352.356} C_DIS
LIN {X 0.273,Y -557.584,Z 1110.754,A 0.000,B 0.000,C 90.000,E1 351.659} C_DIS
LIN {X 0.215,Y -560.880,Z 1110.750,A 0.000,B 0.000,C 90.000,E1 350.971} C_DIS
LIN {X -0.039,Y -563.349,Z 1110.747,A 0.000,B 0.000,C 90.000,E1 350.443} C_DIS
LIN {X 0.283,Y -565.690,Z 1110.744,A 0.000,B 0.000,C 90.000,E1 349.859} C_DIS
LIN {X -0.246,Y -569.944,Z 1110.738,A 0.000,B 0.000,C 90.000,E1 348.814} C_DIS
LIN {X -0.245,Y -572.909,Z 1110.733,A 0.000,B 0.000,C 90.000,E1 347.993} C_DIS
LIN {X -0.009,Y -576.555,Z 1110.727,A 0.000,B 0.000,C 90.000,E1 346.881} C_DIS
LIN {X -0.147,Y -579.862,Z 1110.721,A 0.000,B 0.000,C 90.000,E1 345.811} C_DIS
LIN {X -0.003,Y -583.869,Z 1110.714,A 0.000,B 0.000,C 90.000,E1 344.448} C_DIS
LIN {X 0.128,Y -586.175,Z 1110.709,A 0.000,B 0.000,C 90.000,E1 343.630} C_DIS
LIN {X -0.031,Y -589.869,Z 1110.702,A 0.000,B 0.000,C 90.000,E1 342.308} C_DIS
LIN {X 0.187,Y -592.594,Z 1110.696,A 0.000,B 0.000,C 90.000,E1 341.221} C_DIS
LIN {X -0.225,Y -595.780,Z 1110.688,A 0.000,B 0.000,C 90.000,E1 339.934} C_DIS
LIN {X -0.177,Y -597.500,Z 1110.684,A 0.000,B 0.000,C 90.000,E1 339.135} C_DIS
LIN {X -0.111,Y -599.031,Z 1110.680,A 0.000,B 0.000,C 90.000,E1 338.337} C_DIS
LIN {X 0.134,Y -601.225,Z 1110.672,A 0.000,B 0.000,C 90.000,E1 336.997} C_DIS
LIN {X -0.086,Y -602.328,Z 1110.668,A 0.000,B 0.000,C 90.000,E1 336.230} C_DIS
LIN {X -0.051,Y -603.523,Z 1110.662,A 0.000,B 0.000,C 90.000,E1 335.177} C_DIS
LIN {X -0.299,Y -604.543,Z 1110.656,A 0.000,B 0.000,C 90.000,E1 334.152} C_DIS
LIN {X -0.046,Y -605.243,Z 1110.649,A 0.000,B 0.000,C 90.000,E1 332.820} C_DIS
LIN {X 0.121,Y -605.413,Z 1110.646,A 0.000,B 0.000,C 90.000,E1 332.281} C_DIS
LIN {X -0.102,Y -605.400,Z 1110.640,A 0.000,B 0.000,C 90.000,E1 331.257} C_DIS
LIN {X 0.019,Y -604.946,Z 1110.636,A 0.000,B 0.000,C 90.000,E1 330.461} C_DIS
LIN {X -0.102,Y -604.554,Z 1110.633,A 0.000,B 0.000,C 90.000,E1 329.950} C_DIS
LIN {X 0.008,Y -603.561,Z 1110.629,A 0.000,B 0.000,C 90.000,E1 329.154} C_DIS
LIN {X -0.164,Y -601.589,Z 1110.623,A 0.000,B 0.000,C 90.000,E1 328.122} C_DIS
LIN {X -0.085,Y -599.800,Z 1110.619,A 0.000,B 0.000,C 90.000,E1 327.327} C_DIS
LIN {X -0.300,Y -596.867,Z 1110.613,A 0.000,B 0.000,C 90.000,E1 326.294} C_DIS
LIN {X 0.159,Y -595.266,Z 1110.610,A 0.000,B 0.000,C 90.000,E1 325.722} C_DIS
LIN {X -0.116,Y -591.632,Z 1110.604,A 0.000,B 0.000,C 90.000,E1 324.689} C_DIS
LIN {X -0.100,Y -587.829,Z 1110.598,A 0.000,B 0.000,C 90.000,E1 323.623} C_DIS
LIN {X -0.138,Y -583.773,Z 1110.592,A 0.000,B 0.000,C 90.000,E1 322.557} C_DIS
LIN {X 0.121,Y -579.541,Z 1110.586,A 0.000,B 0.000,C 90.000,E1 321.457} C_DIS
LIN {X 0.002,Y -577.132,Z 1110.583,A 0.000,B 0.000,C 90.000,E1 320.928} C_DIS
LIN {X 0.315,Y -574.898,Z 1110.580,A 0.000,B 0.000,C 90.000,E1 320.356} C_DIS
LIN {X -0.120,Y -569.451,Z 1110.573,A 0.000,B 0.000,C 90.000,E1 319.175} C_DIS
LIN {X -0.178,Y -567.404,Z 1110.571,A 0.000,B 0.000,C 90.000,E1 318.771} C_DIS
LIN {X -0.041,Y -562.123,Z 1110.566,A 0.000,B 0.000,C 90.000,E1 317.796} C_DIS
LIN {X -0.052,Y -557.963,Z 1110.562,A 0.000,B 0.000,C 90.000,E1 317.106} C_DIS
LIN {X -0.288,Y -552.247,Z 1110.557,A 0.000,B 0.000,C 90.000,E1 316.296} C_DIS
LIN {X 0.031,Y -543.560,Z 1110.550,A 0.000,B 0.000,C 90.000,E1 315.000} C_DIS
LIN {X -0.149,Y -540.881,Z 1110.548,A 0.000,B 0.000,C 90.000,E1 314.595} C_DIS
LIN {X -0.001,Y -537.790,Z 1110.545,A 0.000,B 0.000,C 90.000,E1 314.028} C_DIS
LIN {X -0.043,Y -534.270,Z 1110.540,A 0.000,B 0.000,C 90.000,E1 313.176} C_DIS
LIN {X -0.082,Y -533.465,Z 1110.538,A 0.000,B 0.000,C 90.000,E1 312.894} C_DIS
LIN {X -0.113,Y -532.167,Z 1110.535,A 0.000,B 0.000,C 90.000,E1 312.324} C_DIS
LIN {X 0.057,Y -531.705,Z 1110.534,A 0.000,B 0.000,C 90.000,E1 312.162} C_DIS
LIN {X 0.106,Y -530.380,Z 1110.529,A 0.000,B 0.000,C 90.000,E1 311.229} C_DIS
LIN {X -0.035,Y -529.602,Z 1110.523,A 0.000,B 0.000,C 90.000,E1 310.092} C_DIS
LIN {X -0.235,Y -529.591,Z 1110.513,A 0.000,B 0.000,C 90.000,E1 308.382} C_DIS
LIN {X -0.272,Y -529.773,Z 1110.510,A 0.000,B 0.000,C 90.000,E1 307.810} C_DIS
LIN {X -0.016,Y -531.373,Z 1110.492,A 0.000,B 0.000,C 90.000,E1 304.612} C_DIS
LIN {X 0.042,Y -532.458,Z 1110.483,A 0.000,B 0.000,C 90.000,E1 302.880} C_DIS
LIN {X -0.010,Y -534.001,Z 1110.472,A 0.000,B 0.000,C 90.000,E1 300.875} C_DIS
LIN {X -0.185,Y -535.023,Z 1110.464,A 0.000,B 0.000,C 90.000,E1 299.461} C_DIS
LIN {X 0.162,Y -535.651,Z 1110.459,A 0.000,B 0.000,C 90.000,E1 298.565} C_DIS
LIN {X -0.062,Y -536.551,Z 1110.449,A 0.000,B 0.000,C 90.000,E1 296.873} C_DIS
LIN {X -0.173,Y -536.918,Z 1110.445,A 0.000,B 0.000,C 90.000,E1 296.027} C_DIS
LIN {X -0.094,Y -537.364,Z 1110.437,A 0.000,B 0.000,C 90.000,E1 294.591} C_DIS
LIN {X 0.005,Y -537.664,Z 1110.429,A 0.000,B 0.000,C 90.000,E1 293.153} C_DIS
LIN {X 0.105,Y -537.809,Z 1110.421,A 0.000,B 0.000,C 90.000,E1 291.716} C_DIS
LIN {X -0.218,Y -537.871,Z 1110.414,A 0.000,B 0.000,C 90.000,E1 290.610} C_DIS
LIN {X -0.037,Y -537.788,Z 1110.408,A 0.000,B 0.000,C 90.000,E1 289.450} C_DIS
LIN {X -0.286,Y -537.454,Z 1110.399,A 0.000,B 0.000,C 90.000,E1 287.764} C_DIS
LIN {X -0.079,Y -537.075,Z 1110.391,A 0.000,B 0.000,C 90.000,E1 286.315} C_DIS
LIN {X -0.236,Y -536.696,Z 1110.384,A 0.000,B 0.000,C 90.000,E1 285.190} C_DIS
LIN {X 0.182,Y -536.015,Z 1110.376,A 0.000,B 0.000,C 90.000,E1 283.716} C_DIS
LIN {X 0.178,Y -535.055,Z 1110.365,A 0.000,B 0.000,C 90.000,E1 281.715} C_DIS
LIN {X 0.024,Y -534.033,Z 1110.354,A 0.000,B 0.000,C 90.000,E1 279.726} C_DIS
LIN {X 0.186,Y -533.041,Z 1110.343,A 0.000,B 0.000,C 90.000,E1 277.701} C_DIS
LIN {X 0.252,Y -532.343,Z 1110.335,A 0.000,B 0.000,C 90.000,E1 276.258} C_DIS
LIN {X -0.254,Y -531.502,Z 1110.325,A 0.000,B 0.000,C 90.000,E1 274.588} C_DIS
LIN {X 0.237,Y -530.752,Z 1110.316,A 0.000,B 0.000,C 90.000,E1 272.808} C_DIS
LIN {X 0.137,Y -529.813,Z 1110.305,A 0.000,B 0.000,C 90.000,E1 270.802} C_DIS
LIN {X 0.047,Y -529.149,Z 1110.297,A 0.000,B 0.000,C 90.000,E1 269.370} C_DIS
LIN {X -0.044,Y -528.434,Z 1110.289,A 0.000,B 0.000,C 90.000,E1 267.936} C_DIS
LIN {X -0.145,Y -527.560,Z 1110.281,A 0.000,B 0.000,C 90.000,E1 266.502} C_DIS
LIN {X -0.269,Y -526.479,Z 1110.271,A 0.000,B 0.000,C 90.000,E1 264.780} C_DIS
LIN {X 0.186,Y -525.614,Z 1110.264,A 0.000,B 0.000,C 90.000,E1 263.571} C_DIS
LIN {X 0.168,Y -524.520,Z 1110.258,A 0.000,B 0.000,C 90.000,E1 262.413} C_DIS
LIN {X 0.101,Y -521.903,Z 1110.243,A 0.000,B 0.000,C 90.000,E1 259.803} C_DIS
LIN {X 0.130,Y -520.250,Z 1110.234,A 0.000,B 0.000,C 90.000,E1 258.049} C_DIS
LIN {X 0.114,Y -518.582,Z 1110.224,A 0.000,B 0.000,C 90.000,E1 256.297} C_DIS
LIN {X -0.306,Y -517.484,Z 1110.218,A 0.000,B 0.000,C 90.000,E1 255.172} C_DIS
LIN {X -0.125,Y -515.911,Z 1110.209,A 0.000,B 0.000,C 90.000,E1 253.685} C_DIS
LIN {X 0.137,Y -514.110,Z 1110.200,A 0.000,B 0.000,C 90.000,E1 251.891} C_DIS
LIN {X 0.081,Y -512.542,Z 1110.191,A 0.000,B 0.000,C 90.000,E1 250.423} C_DIS
LIN {X 0.043,Y -510.141,Z 1110.180,A 0.000,B 0.000,C 90.000,E1 248.358} C_DIS
LIN {X 0.103,Y -508.339,Z 1110.172,A 0.000,B 0.000,C 90.000,E1 246.869} C_DIS
LIN {X 0.141,Y -507.090,Z 1110.167,A 0.000,B 0.000,C 90.000,E1 245.973} C_DIS
LIN {X 0.138,Y -504.941,Z 1110.158,A 0.000,B 0.000,C 90.000,E1 244.485} C_DIS
LIN {X -0.004,Y -503.049,Z 1110.152,A 0.000,B 0.000,C 90.000,E1 243.307} C_DIS
LIN {X -0.038,Y -500.160,Z 1110.142,A 0.000,B 0.000,C 90.000,E1 241.513} C_DIS
LIN {X 0.050,Y -497.631,Z 1110.133,A 0.000,B 0.000,C 90.000,E1 239.999} C_DIS
LIN {X 0.067,Y -495.677,Z 1110.127,A 0.000,B 0.000,C 90.000,E1 238.791} C_DIS
LIN {X -0.095,Y -492.999,Z 1110.118,A 0.000,B 0.000,C 90.000,E1 237.296} C_DIS
LIN {X 0.099,Y -490.375,Z 1110.110,A 0.000,B 0.000,C 90.000,E1 235.754} C_DIS
LIN {X -0.137,Y -488.186,Z 1110.103,A 0.000,B 0.000,C 90.000,E1 234.562} C_DIS
LIN {X 0.102,Y -485.321,Z 1110.095,A 0.000,B 0.000,C 90.000,E1 233.004} C_DIS
LIN {X 0.197,Y -482.372,Z 1110.086,A 0.000,B 0.000,C 90.000,E1 231.457} C_DIS
LIN {X -0.243,Y -479.986,Z 1110.079,A 0.000,B 0.000,C 90.000,E1 230.275} C_DIS
LIN {X 0.064,Y -476.954,Z 1110.071,A 0.000,B 0.000,C 90.000,E1 228.690} C_DIS
LIN {X -0.173,Y -472.814,Z 1110.058,A 0.000,B 0.000,C 90.000,E1 226.539} C_DIS
LIN {X 0.036,Y -469.362,Z 1110.048,A 0.000,B 0.000,C 90.000,E1 224.636} C_DIS
LIN {X 0.094,Y -466.571,Z 1110.039,A 0.000,B 0.000,C 90.000,E1 223.056} C_DIS
LIN {X 0.188,Y -463.323,Z 1110.029,A 0.000,B 0.000,C 90.000,E1 221.148} C_DIS
LIN {X -0.056,Y -459.774,Z 1110.016,A 0.000,B 0.000,C 90.000,E1 218.955} C_DIS
LIN {X 0.027,Y -456.343,Z 1110.004,A 0.000,B 0.000,C 90.000,E1 216.710} C_DIS
LIN {X 0.037,Y -454.023,Z 1109.995,A 0.000,B 0.000,C 90.000,E1 215.105} C_DIS
LIN {X 0.006,Y -451.722,Z 1109.986,A 0.000,B 0.000,C 90.000,E1 213.499} C_DIS
LIN {X -0.163,Y -448.660,Z 1109.974,A 0.000,B 0.000,C 90.000,E1 211.258} C_DIS
LIN {X 0.126,Y -445.892,Z 1109.961,A 0.000,B 0.000,C 90.000,E1 208.949} C_DIS
LIN {X 0.121,Y -443.621,Z 1109.948,A 0.000,B 0.000,C 90.000,E1 206.668} C_DIS
LIN {X -0.129,Y -442.874,Z 1109.943,A 0.000,B 0.000,C 90.000,E1 205.720} C_DIS
LIN {X 0.053,Y -442.198,Z 1109.936,A 0.000,B 0.000,C 90.000,E1 204.387} C_DIS
LIN {X 0.044,Y -442.361,Z 1109.928,A 0.000,B 0.000,C 90.000,E1 203.078} C_DIS
LIN {X 0.038,Y -443.303,Z 1109.921,A 0.000,B 0.000,C 90.000,E1 201.770} C_DIS
LIN {X 0.165,Y -444.034,Z 1109.917,A 0.000,B 0.000,C 90.000,E1 201.099} C_DIS
LIN {X 0.161,Y -445.905,Z 1109.912,A 0.000,B 0.000,C 90.000,E1 200.120} C_DIS
LIN {X 0.176,Y -448.223,Z 1109.906,A 0.000,B 0.000,C 90.000,E1 199.141} C_DIS
LIN {X -0.052,Y -451.930,Z 1109.899,A 0.000,B 0.000,C 90.000,E1 197.873} C_DIS
LIN {X 0.071,Y -459.718,Z 1109.887,A 0.000,B 0.000,C 90.000,E1 195.607} C_DIS
LIN {X 0.126,Y -469.669,Z 1109.873,A 0.000,B 0.000,C 90.000,E1 193.063} C_DIS
LIN {X 0.084,Y -479.664,Z 1109.860,A 0.000,B 0.000,C 90.000,E1 190.725} C_DIS
LIN {X 0.080,Y -487.174,Z 1109.850,A 0.000,B 0.000,C 90.000,E1 189.029} C_DIS
LIN {X 0.019,Y -492.622,Z 1109.844,A 0.000,B 0.000,C 90.000,E1 187.814} C_DIS
LIN {X -0.021,Y -498.002,Z 1109.837,A 0.000,B 0.000,C 90.000,E1 186.606} C_DIS
LIN {X -0.050,Y -504.477,Z 1109.828,A 0.000,B 0.000,C 90.000,E1 185.106} C_DIS
LIN {X -0.099,Y -512.361,Z 1109.818,A 0.000,B 0.000,C 90.000,E1 183.326} C_DIS
LIN {X 0.022,Y -520.148,Z 1109.809,A 0.000,B 0.000,C 90.000,E1 181.547} C_DIS
LIN {X 0.074,Y -526.114,Z 1109.801,A 0.000,B 0.000,C 90.000,E1 180.229} C_DIS
LIN {X -0.047,Y -532.632,Z 1109.793,A 0.000,B 0.000,C 90.000,E1 178.797} C_DIS
LIN {X -0.039,Y -539.163,Z 1109.785,A 0.000,B 0.000,C 90.000,E1 177.364} C_DIS
LIN {X -0.135,Y -546.289,Z 1109.777,A 0.000,B 0.000,C 90.000,E1 175.812} C_DIS
LIN {X 0.161,Y -552.667,Z 1109.769,A 0.000,B 0.000,C 90.000,E1 174.375} C_DIS
LIN {X 0.147,Y -560.392,Z 1109.760,A 0.000,B 0.000,C 90.000,E1 172.704} C_DIS
LIN {X -0.125,Y -566.117,Z 1109.753,A 0.000,B 0.000,C 90.000,E1 171.489} C_DIS
LIN {X 0.303,Y -573.489,Z 1109.744,A 0.000,B 0.000,C 90.000,E1 169.803} C_DIS
LIN {X -0.233,Y -578.937,Z 1109.737,A 0.000,B 0.000,C 90.000,E1 168.634} C_DIS
LIN {X -0.129,Y -582.432,Z 1109.732,A 0.000,B 0.000,C 90.000,E1 167.813} C_DIS
LIN {X 0.252,Y -586.975,Z 1109.726,A 0.000,B 0.000,C 90.000,E1 166.700} C_DIS
LIN {X 0.120,Y -591.286,Z 1109.720,A 0.000,B 0.000,C 90.000,E1 165.644} C_DIS
LIN {X 0.189,Y -595.369,Z 1109.714,A 0.000,B 0.000,C 90.000,E1 164.574} C_DIS
LIN {X 0.027,Y -600.138,Z 1109.707,A 0.000,B 0.000,C 90.000,E1 163.268} C_DIS
LIN {X -0.082,Y -602.838,Z 1109.703,A 0.000,B 0.000,C 90.000,E1 162.489} C_DIS
LIN {X 0.244,Y -607.063,Z 1109.695,A 0.000,B 0.000,C 90.000,E1 161.148} C_DIS
LIN {X 0.143,Y -610.252,Z 1109.690,A 0.000,B 0.000,C 90.000,E1 160.115} C_DIS
LIN {X 0.081,Y -613.304,Z 1109.684,A 0.000,B 0.000,C 90.000,E1 159.082} C_DIS
LIN {X 0.019,Y -616.837,Z 1109.677,A 0.000,B 0.000,C 90.000,E1 157.794} C_DIS
LIN {X 0.248,Y -620.310,Z 1109.670,A 0.000,B 0.000,C 90.000,E1 156.485} C_DIS
LIN {X -0.030,Y -623.642,Z 1109.662,A 0.000,B 0.000,C 90.000,E1 155.229} C_DIS
LIN {X 0.000,Y -626.189,Z 1109.657,A 0.000,B 0.000,C 90.000,E1 154.204} C_DIS
LIN {X 0.092,Y -629.260,Z 1109.650,A 0.000,B 0.000,C 90.000,E1 152.922} C_DIS
LIN {X -0.260,Y -633.206,Z 1109.640,A 0.000,B 0.000,C 90.000,E1 151.179} C_DIS
LIN {X 0.238,Y -635.922,Z 1109.633,A 0.000,B 0.000,C 90.000,E1 149.871} C_DIS
LIN {X 0.226,Y -638.531,Z 1109.626,A 0.000,B 0.000,C 90.000,E1 148.614} C_DIS
LIN {X 0.049,Y -641.026,Z 1109.619,A 0.000,B 0.000,C 90.000,E1 147.375} C_DIS
LIN {X -0.029,Y -643.908,Z 1109.610,A 0.000,B 0.000,C 90.000,E1 145.881} C_DIS
LIN {X 0.254,Y -646.121,Z 1109.604,A 0.000,B 0.000,C 90.000,E1 144.609} C_DIS
LIN {X 0.020,Y -649.194,Z 1109.594,A 0.000,B 0.000,C 90.000,E1 142.889} C_DIS
LIN {X 0.295,Y -652.759,Z 1109.583,A 0.000,B 0.000,C 90.000,E1 140.884} C_DIS
LIN {X 0.048,Y -656.450,Z 1109.572,A 0.000,B 0.000,C 90.000,E1 138.933} C_DIS
LIN {X -0.106,Y -659.335,Z 1109.564,A 0.000,B 0.000,C 90.000,E1 137.472} C_DIS
LIN {X 0.208,Y -663.968,Z 1109.552,A 0.000,B 0.000,C 90.000,E1 135.243} C_DIS
LIN {X 0.184,Y -669.048,Z 1109.539,A 0.000,B 0.000,C 90.000,E1 133.056} C_DIS
LIN {X -0.128,Y -674.389,Z 1109.527,A 0.000,B 0.000,C 90.000,E1 130.906} C_DIS
LIN {X 0.148,Y -677.934,Z 1109.519,A 0.000,B 0.000,C 90.000,E1 129.439} C_DIS
LIN {X -0.421,Y -682.254,Z 1109.510,A 0.000,B 0.000,C 90.000,E1 127.810} C_DIS
LIN {X -0.023,Y -685.321,Z 1109.503,A 0.000,B 0.000,C 90.000,E1 126.583} C_DIS
LIN {X -0.195,Y -687.124,Z 1109.499,A 0.000,B 0.000,C 90.000,E1 125.884} C_DIS
LIN {X -0.094,Y -690.622,Z 1109.491,A 0.000,B 0.000,C 90.000,E1 124.452} C_DIS
LIN {X -0.135,Y -694.093,Z 1109.484,A 0.000,B 0.000,C 90.000,E1 123.038} C_DIS
LIN {X -0.337,Y -696.898,Z 1109.477,A 0.000,B 0.000,C 90.000,E1 121.878} C_DIS
LIN {X -0.164,Y -698.883,Z 1109.472,A 0.000,B 0.000,C 90.000,E1 120.924} C_DIS
LIN {X -0.327,Y -700.626,Z 1109.467,A 0.000,B 0.000,C 90.000,E1 120.001} C_DIS
LIN {X -0.192,Y -702.536,Z 1109.460,A 0.000,B 0.000,C 90.000,E1 118.821} C_DIS
LIN {X 0.310,Y -703.820,Z 1109.455,A 0.000,B 0.000,C 90.000,E1 117.847} C_DIS
LIN {X -0.086,Y -704.599,Z 1109.451,A 0.000,B 0.000,C 90.000,E1 117.180} C_DIS
LIN {X 0.061,Y -705.670,Z 1109.443,A 0.000,B 0.000,C 90.000,E1 115.771} C_DIS
LIN {X -0.011,Y -705.911,Z 1109.439,A 0.000,B 0.000,C 90.000,E1 115.079} C_DIS
LIN {X 0.275,Y -705.862,Z 1109.437,A 0.000,B 0.000,C 90.000,E1 114.591} C_DIS
LIN {X -0.077,Y -705.158,Z 1109.434,A 0.000,B 0.000,C 90.000,E1 114.155} C_DIS
LIN {X 0.211,Y -704.694,Z 1109.433,A 0.000,B 0.000,C 90.000,E1 113.898} C_DIS
LIN {X -0.005,Y -702.309,Z 1109.430,A 0.000,B 0.000,C 90.000,E1 113.334} C_DIS
LIN {X 0.135,Y -701.536,Z 1109.429,A 0.000,B 0.000,C 90.000,E1 113.206} C_DIS
LIN {X -0.127,Y -697.448,Z 1109.427,A 0.000,B 0.000,C 90.000,E1 112.770} C_DIS
LIN {X 0.002,Y -696.114,Z 1109.426,A 0.000,B 0.000,C 90.000,E1 112.642} C_DIS
LIN {X 0.131,Y -693.948,Z 1109.425,A 0.000,B 0.000,C 90.000,E1 112.514} C_DIS
LIN {X 0.216,Y -686.533,Z 1109.423,A 0.000,B 0.000,C 90.000,E1 112.206} C_DIS
LIN {X 0.203,Y -684.474,Z 1109.423,A 0.000,B 0.000,C 90.000,E1 112.153} C_DIS
LIN {X 0.025,Y -676.406,Z 1109.423,A 0.000,B 0.000,C 90.000,E1 112.078} C_DIS
LIN {X -0.026,Y -603.843,Z 1109.423,A 0.000,B 0.000,C 90.000,E1 112.078} C_DIS
LIN {X -0.255,Y -600.301,Z 1109.422,A 0.000,B 0.000,C 90.000,E1 111.897} C_DIS
LIN {X 0.221,Y -595.913,Z 1109.420,A 0.000,B 0.000,C 90.000,E1 111.535} C_DIS
LIN {X 0.216,Y -586.596,Z 1109.415,A 0.000,B 0.000,C 90.000,E1 110.737} C_DIS
LIN {X -0.317,Y -578.313,Z 1109.411,A 0.000,B 0.000,C 90.000,E1 110.066} C_DIS
LIN {X -0.073,Y -574.022,Z 1109.409,A 0.000,B 0.000,C 90.000,E1 109.685} C_DIS
LIN {X 0.159,Y -567.961,Z 1109.407,A 0.000,B 0.000,C 90.000,E1 109.214} C_DIS
LIN {X -0.128,Y -561.489,Z 1109.405,A 0.000,B 0.000,C 90.000,E1 108.833} C_DIS
LIN {X 0.318,Y -555.104,Z 1109.403,A 0.000,B 0.000,C 90.000,E1 108.417} C_DIS
LIN {X -0.121,Y -550.104,Z 1109.401,A 0.000,B 0.000,C 90.000,E1 108.109} C_DIS
LIN {X 0.138,Y -548.695,Z 1109.399,A 0.000,B 0.000,C 90.000,E1 107.873} C_DIS
LIN {X 0.096,Y -548.682,Z 1109.399,A 0.000,B 0.000,C 90.000,E1 107.873} C_DIS
LIN {X 0.220,Y -548.357,Z 1109.397,A 0.000,B 0.000,C 90.000,E1 107.457} C_DIS
LIN {X -0.131,Y -548.683,Z 1109.393,A 0.000,B 0.000,C 90.000,E1 106.732} C_DIS
LIN {X -0.122,Y -549.483,Z 1109.387,A 0.000,B 0.000,C 90.000,E1 105.607} C_DIS
LIN {X 0.051,Y -551.400,Z 1109.373,A 0.000,B 0.000,C 90.000,E1 103.063} C_DIS
LIN {X -0.203,Y -553.130,Z 1109.362,A 0.000,B 0.000,C 90.000,E1 101.130} C_DIS
LIN {X -0.100,Y -554.770,Z 1109.352,A 0.000,B 0.000,C 90.000,E1 99.443} C_DIS
LIN {X 0.034,Y -556.490,Z 1109.343,A 0.000,B 0.000,C 90.000,E1 97.757} C_DIS
LIN {X -0.016,Y -557.870,Z 1109.335,A 0.000,B 0.000,C 90.000,E1 96.372} C_DIS
LIN {X -0.174,Y -558.972,Z 1109.329,A 0.000,B 0.000,C 90.000,E1 95.277} C_DIS
LIN {X -0.240,Y -560.125,Z 1109.322,A 0.000,B 0.000,C 90.000,E1 93.898} C_DIS
LIN {X 0.239,Y -561.115,Z 1109.314,A 0.000,B 0.000,C 90.000,E1 92.465} C_DIS
LIN {X 0.277,Y -562.076,Z 1109.305,A 0.000,B 0.000,C 90.000,E1 90.802} C_DIS
LIN {X 0.221,Y -562.785,Z 1109.297,A 0.000,B 0.000,C 90.000,E1 89.427} C_DIS
LIN {X -0.269,Y -563.618,Z 1109.288,A 0.000,B 0.000,C 90.000,E1 87.822} C_DIS
LIN {X 0.279,Y -564.244,Z 1109.280,A 0.000,B 0.000,C 90.000,E1 86.388} C_DIS
LIN {X 0.162,Y -564.725,Z 1109.274,A 0.000,B 0.000,C 90.000,E1 85.298} C_DIS
LIN {X 0.253,Y -565.280,Z 1109.266,A 0.000,B 0.000,C 90.000,E1 83.913} C_DIS
LIN {X 0.060,Y -566.018,Z 1109.256,A 0.000,B 0.000,C 90.000,E1 82.008} C_DIS
LIN {X -0.042,Y -566.693,Z 1109.245,A 0.000,B 0.000,C 90.000,E1 80.095} C_DIS
LIN {X -0.214,Y -567.399,Z 1109.236,A 0.000,B 0.000,C 90.000,E1 78.465} C_DIS
LIN {X -0.264,Y -568.203,Z 1109.227,A 0.000,B 0.000,C 90.000,E1 76.825} C_DIS
LIN {X -0.219,Y -569.407,Z 1109.214,A 0.000,B 0.000,C 90.000,E1 74.629} C_DIS
LIN {X 0.201,Y -571.165,Z 1109.201,A 0.000,B 0.000,C 90.000,E1 72.127} C_DIS
LIN {X 0.308,Y -572.889,Z 1109.189,A 0.000,B 0.000,C 90.000,E1 69.934} C_DIS
LIN {X 0.109,Y -574.128,Z 1109.181,A 0.000,B 0.000,C 90.000,E1 68.592} C_DIS
LIN {X -0.021,Y -575.630,Z 1109.172,A 0.000,B 0.000,C 90.000,E1 66.975} C_DIS
LIN {X -0.273,Y -577.230,Z 1109.162,A 0.000,B 0.000,C 90.000,E1 65.101} C_DIS
LIN {X 0.032,Y -578.283,Z 1109.154,A 0.000,B 0.000,C 90.000,E1 63.717} C_DIS
LIN {X -0.053,Y -579.453,Z 1109.145,A 0.000,B 0.000,C 90.000,E1 62.103} C_DIS
LIN {X 0.025,Y -580.684,Z 1109.135,A 0.000,B 0.000,C 90.000,E1 60.205} C_DIS
LIN {X -0.095,Y -581.473,Z 1109.127,A 0.000,B 0.000,C 90.000,E1 58.869} C_DIS
LIN {X -0.057,Y -582.148,Z 1109.121,A 0.000,B 0.000,C 90.000,E1 57.788} C_DIS
LIN {X 0.184,Y -583.075,Z 1109.111,A 0.000,B 0.000,C 90.000,E1 55.881} C_DIS
LIN {X 0.107,Y -583.881,Z 1109.102,A 0.000,B 0.000,C 90.000,E1 54.276} C_DIS
LIN {X -0.078,Y -584.480,Z 1109.093,A 0.000,B 0.000,C 90.000,E1 52.683} C_DIS
LIN {X -0.342,Y -584.796,Z 1109.088,A 0.000,B 0.000,C 90.000,E1 51.904} C_DIS
LIN {X -0.244,Y -584.947,Z 1109.084,A 0.000,B 0.000,C 90.000,E1 51.090} C_DIS
LIN {X -0.144,Y -585.036,Z 1109.079,A 0.000,B 0.000,C 90.000,E1 50.275} C_DIS
LIN {X -0.127,Y -584.927,Z 1109.072,A 0.000,B 0.000,C 90.000,E1 48.933} C_DIS
LIN {X 0.095,Y -584.736,Z 1109.066,A 0.000,B 0.000,C 90.000,E1 47.838} C_DIS
LIN {X -0.081,Y -584.420,Z 1109.060,A 0.000,B 0.000,C 90.000,E1 46.782} C_DIS
LIN {X 0.276,Y -583.860,Z 1109.052,A 0.000,B 0.000,C 90.000,E1 45.405} C_DIS
LIN {X 0.064,Y -583.214,Z 1109.047,A 0.000,B 0.000,C 90.000,E1 44.352} C_DIS
LIN {X -0.161,Y -582.357,Z 1109.041,A 0.000,B 0.000,C 90.000,E1 43.299} C_DIS
LIN {X 0.019,Y -581.266,Z 1109.035,A 0.000,B 0.000,C 90.000,E1 42.204} C_DIS
LIN {X -0.041,Y -579.532,Z 1109.027,A 0.000,B 0.000,C 90.000,E1 40.862} C_DIS
LIN {X 0.376,Y -578.450,Z 1109.023,A 0.000,B 0.000,C 90.000,E1 40.011} C_DIS
LIN {X -0.093,Y -576.130,Z 1109.015,A 0.000,B 0.000,C 90.000,E1 38.705} C_DIS
LIN {X -0.085,Y -574.533,Z 1109.010,A 0.000,B 0.000,C 90.000,E1 37.890} C_DIS
LIN {X -0.099,Y -572.672,Z 1109.006,A 0.000,B 0.000,C 90.000,E1 37.076} C_DIS
LIN {X -0.018,Y -570.606,Z 1109.001,A 0.000,B 0.000,C 90.000,E1 36.251} C_DIS
LIN {X -0.211,Y -569.015,Z 1108.998,A 0.000,B 0.000,C 90.000,E1 35.724} C_DIS
LIN {X 0.041,Y -567.261,Z 1108.995,A 0.000,B 0.000,C 90.000,E1 35.152} C_DIS
LIN {X 0.070,Y -564.419,Z 1108.991,A 0.000,B 0.000,C 90.000,E1 34.326} C_DIS
LIN {X -0.031,Y -562.245,Z 1108.988,A 0.000,B 0.000,C 90.000,E1 33.785} C_DIS
LIN {X -0.050,Y -558.724,Z 1108.983,A 0.000,B 0.000,C 90.000,E1 32.959} C_DIS
LIN {X -0.001,Y -555.525,Z 1108.979,A 0.000,B 0.000,C 90.000,E1 32.260} C_DIS
LIN {X 0.244,Y -550.598,Z 1108.974,A 0.000,B 0.000,C 90.000,E1 31.258} C_DIS
LIN {X -0.199,Y -545.997,Z 1108.969,A 0.000,B 0.000,C 90.000,E1 30.463} C_DIS
LIN {X -0.076,Y -540.330,Z 1108.964,A 0.000,B 0.000,C 90.000,E1 29.461} C_DIS
LIN {X -0.014,Y -535.841,Z 1108.960,A 0.000,B 0.000,C 90.000,E1 28.743} C_DIS
LIN {X 0.150,Y -531.892,Z 1108.957,A 0.000,B 0.000,C 90.000,E1 28.153} C_DIS
LIN {X 0.038,Y -527.711,Z 1108.953,A 0.000,B 0.000,C 90.000,E1 27.590} C_DIS
LIN {X -0.016,Y -522.166,Z 1108.949,A 0.000,B 0.000,C 90.000,E1 26.873} C_DIS
LIN {X -0.025,Y -518.596,Z 1108.947,A 0.000,B 0.000,C 90.000,E1 26.437} C_DIS
LIN {X 0.008,Y -513.533,Z 1108.944,A 0.000,B 0.000,C 90.000,E1 25.848} C_DIS
LIN {X -0.292,Y -506.968,Z 1108.940,A 0.000,B 0.000,C 90.000,E1 25.155} C_DIS
LIN {X -0.110,Y -496.314,Z 1108.933,A 0.000,B 0.000,C 90.000,E1 24.027} C_DIS
LIN {X -0.010,Y -483.872,Z 1108.927,A 0.000,B 0.000,C 90.000,E1 22.823} C_DIS
LIN {X -0.187,Y -478.367,Z 1108.924,A 0.000,B 0.000,C 90.000,E1 22.333} C_DIS
LIN {X 0.114,Y -472.377,Z 1108.921,A 0.000,B 0.000,C 90.000,E1 21.770} C_DIS
LIN {X -0.003,Y -458.997,Z 1108.915,A 0.000,B 0.000,C 90.000,E1 20.610} C_DIS
LIN {X 0.144,Y -435.302,Z 1108.902,A 0.000,B 0.000,C 90.000,E1 18.417} C_DIS
LIN {X -0.074,Y -421.130,Z 1108.894,A 0.000,B 0.000,C 90.000,E1 16.985} C_DIS
LIN {X 0.123,Y -410.374,Z 1108.887,A 0.000,B 0.000,C 90.000,E1 15.717} C_DIS
LIN {X -0.069,Y -400.075,Z 1108.880,A 0.000,B 0.000,C 90.000,E1 14.411} C_DIS
LIN {X 0.126,Y -396.261,Z 1108.877,A 0.000,B 0.000,C 90.000,E1 13.772} C_DIS
LIN {X -0.082,Y -394.481,Z 1108.875,A 0.000,B 0.000,C 90.000,E1 13.411} C_DIS
LIN {X -0.144,Y -393.743,Z 1108.874,A 0.000,B 0.000,C 90.000,E1 13.244} C_DIS
LIN {X 0.149,Y -392.414,Z 1108.870,A 0.000,B 0.000,C 90.000,E1 12.647} C_DIS
LIN {X 0.057,Y -392.035,Z 1108.866,A 0.000,B 0.000,C 90.000,E1 11.951} C_DIS
LIN {X 0.028,Y -392.479,Z 1108.864,A 0.000,B 0.000,C 90.000,E1 11.422} C_DIS
LIN {X -0.069,Y -394.836,Z 1108.856,A 0.000,B 0.000,C 90.000,E1 10.018} C_DIS
LIN {X 0.189,Y -397.813,Z 1108.848,A 0.000,B 0.000,C 90.000,E1 8.568} C_DIS
LIN {X 0.037,Y -402.243,Z 1108.838,A 0.000,B 0.000,C 90.000,E1 6.834} C_DIS
LIN {X -0.032,Y -404.826,Z 1108.832,A 0.000,B 0.000,C 90.000,E1 5.796} C_DIS
LIN {X -0.055,Y -406.410,Z 1108.829,A 0.000,B 0.000,C 90.000,E1 5.277} C_DIS
LIN {X -0.074,Y -407.061,Z 1108.828,A 0.000,B 0.000,C 90.000,E1 5.106} C_DIS
LIN {X -0.057,Y -410.906,Z 1108.825,A 0.000,B 0.000,C 90.000,E1 4.416} C_DIS
LIN {X -0.068,Y -412.156,Z 1108.824,A 0.000,B 0.000,C 90.000,E1 4.245} C_DIS
LIN {X -0.085,Y -417.203,Z 1108.821,A 0.000,B 0.000,C 90.000,E1 3.784} C_DIS
LIN {X 0.068,Y -426.174,Z 1108.818,A 0.000,B 0.000,C 90.000,E1 3.154} C_DIS
LIN {X -0.037,Y -445.889,Z 1108.810,A 0.000,B 0.000,C 90.000,E1 1.835} C_DIS
LIN {X -0.101,Y -465.590,Z 1108.803,A 0.000,B 0.000,C 90.000,E1 0.573} C_DIS
LIN {X -0.205,Y -479.210,Z 1108.798,A 0.000,B 0.000,C 90.000,E1 359.714} C_DIS
LIN {X -0.210,Y -488.807,Z 1108.795,A 0.000,B 0.000,C 90.000,E1 359.083} C_DIS
LIN {X 0.048,Y -498.036,Z 1108.791,A 0.000,B 0.000,C 90.000,E1 358.396} C_DIS
LIN {X 0.216,Y -503.945,Z 1108.789,A 0.000,B 0.000,C 90.000,E1 357.936} C_DIS
LIN {X 0.098,Y -511.286,Z 1108.786,A 0.000,B 0.000,C 90.000,E1 357.364} C_DIS
LIN {X -0.221,Y -517.120,Z 1108.783,A 0.000,B 0.000,C 90.000,E1 356.906} C_DIS
LIN {X 0.203,Y -523.991,Z 1108.779,A 0.000,B 0.000,C 90.000,E1 356.216} C_DIS
LIN {X -0.179,Y -530.539,Z 1108.775,A 0.000,B 0.000,C 90.000,E1 355.584} C_DIS
LIN {X -0.118,Y -535.581,Z 1108.772,A 0.000,B 0.000,C 90.000,E1 355.008} C_DIS
LIN {X -0.224,Y -541.135,Z 1108.768,A 0.000,B 0.000,C 90.000,E1 354.318} C_DIS
LIN {X 0.208,Y -546.208,Z 1108.764,A 0.000,B 0.000,C 90.000,E1 353.571} C_DIS
LIN {X 0.129,Y -550.817,Z 1108.760,A 0.000,B 0.000,C 90.000,E1 352.875} C_DIS
LIN {X 0.275,Y -554.221,Z 1108.757,A 0.000,B 0.000,C 90.000,E1 352.299} C_DIS
LIN {X 0.272,Y -557.941,Z 1108.754,A 0.000,B 0.000,C 90.000,E1 351.602} C_DIS
LIN {X -0.088,Y -560.616,Z 1108.750,A 0.000,B 0.000,C 90.000,E1 351.084} C_DIS
LIN {X -0.281,Y -564.312,Z 1108.746,A 0.000,B 0.000,C 90.000,E1 350.274} C_DIS
LIN {X 0.041,Y -566.605,Z 1108.743,A 0.000,B 0.000,C 90.000,E1 349.690} C_DIS
LIN {X 0.189,Y -570.834,Z 1108.737,A 0.000,B 0.000,C 90.000,E1 348.578} C_DIS
LIN {X 0.202,Y -573.791,Z 1108.732,A 0.000,B 0.000,C 90.000,E1 347.757} C_DIS
LIN {X 0.248,Y -576.537,Z 1108.728,A 0.000,B 0.000,C 90.000,E1 346.937} C_DIS
LIN {X 0.188,Y -580.721,Z 1108.720,A 0.000,B 0.000,C 90.000,E1 345.589} C_DIS
LIN {X -0.227,Y -584.710,Z 1108.713,A 0.000,B 0.000,C 90.000,E1 344.283} C_DIS
LIN {X 0.070,Y -587.037,Z 1108.708,A 0.000,B 0.000,C 90.000,E1 343.449} C_DIS
LIN {X -0.073,Y -590.714,Z 1108.701,A 0.000,B 0.000,C 90.000,E1 342.127} C_DIS
LIN {X 0.158,Y -593.457,Z 1108.695,A 0.000,B 0.000,C 90.000,E1 341.040} C_DIS
LIN {X -0.135,Y -596.016,Z 1108.689,A 0.000,B 0.000,C 90.000,E1 340.007} C_DIS
LIN {X -0.185,Y -598.303,Z 1108.683,A 0.000,B 0.000,C 90.000,E1 338.954} C_DIS
LIN {X -0.111,Y -599.829,Z 1108.679,A 0.000,B 0.000,C 90.000,E1 338.156} C_DIS
LIN {X -0.174,Y -601.963,Z 1108.671,A 0.000,B 0.000,C 90.000,E1 336.847} C_DIS
LIN {X -0.070,Y -603.023,Z 1108.667,A 0.000,B 0.000,C 90.000,E1 336.049} C_DIS
LIN {X 0.224,Y -604.226,Z 1108.661,A 0.000,B 0.000,C 90.000,E1 334.973} C_DIS
LIN {X -0.007,Y -605.244,Z 1108.655,A 0.000,B 0.000,C 90.000,E1 333.948} C_DIS
LIN {X 0.263,Y -605.942,Z 1108.648,A 0.000,B 0.000,C 90.000,E1 332.615} C_DIS
LIN {X 0.101,Y -606.104,Z 1108.644,A 0.000,B 0.000,C 90.000,E1 331.847} C_DIS
LIN {X 0.228,Y -606.064,Z 1108.639,A 0.000,B 0.000,C 90.000,E1 331.051} C_DIS
LIN {X 0.301,Y -605.444,Z 1108.634,A 0.000,B 0.000,C 90.000,E1 329.999} C_DIS
LIN {X -0.094,Y -604.575,Z 1108.629,A 0.000,B 0.000,C 90.000,E1 329.253} C_DIS
LIN {X -0.223,Y -603.765,Z 1108.626,A 0.000,B 0.000,C 90.000,E1 328.742} C_DIS
LIN {X 0.198,Y -602.315,Z 1108.622,A 0.000,B 0.000,C 90.000,E1 327.916} C_DIS
LIN {X -0.221,Y -600.528,Z 1108.618,A 0.000,B 0.000,C 90.000,E1 327.168} C_DIS
LIN {X -0.159,Y -598.470,Z 1108.613,A 0.000,B 0.000,C 90.000,E1 326.373} C_DIS
LIN {X -0.287,Y -596.149,Z 1108.609,A 0.000,B 0.000,C 90.000,E1 325.595} C_DIS
LIN {X 0.055,Y -593.626,Z 1108.604,A 0.000,B 0.000,C 90.000,E1 324.769} C_DIS
LIN {X 0.303,Y -589.116,Z 1108.597,A 0.000,B 0.000,C 90.000,E1 323.417} C_DIS
LIN {X 0.083,Y -586.365,Z 1108.593,A 0.000,B 0.000,C 90.000,E1 322.637} C_DIS
LIN {X 0.100,Y -581.401,Z 1108.585,A 0.000,B 0.000,C 90.000,E1 321.295} C_DIS
LIN {X -0.203,Y -578.434,Z 1108.581,A 0.000,B 0.000,C 90.000,E1 320.517} C_DIS
LIN {X 0.346,Y -573.996,Z 1108.575,A 0.000,B 0.000,C 90.000,E1 319.380} C_DIS
LIN {X -0.230,Y -569.876,Z 1108.569,A 0.000,B 0.000,C 90.000,E1 318.485} C_DIS
LIN {X -0.282,Y -567.898,Z 1108.567,A 0.000,B 0.000,C 90.000,E1 318.081} C_DIS
LIN {X 0.002,Y -563.307,Z 1108.562,A 0.000,B 0.000,C 90.000,E1 317.229} C_DIS
LIN {X 0.231,Y -558.426,Z 1108.558,A 0.000,B 0.000,C 90.000,E1 316.377} C_DIS
LIN {X 0.002,Y -552.729,Z 1108.553,A 0.000,B 0.000,C 90.000,E1 315.567} C_DIS
LIN {X 0.327,Y -544.170,Z 1108.546,A 0.000,B 0.000,C 90.000,E1 314.271} C_DIS
LIN {X -0.035,Y -540.768,Z 1108.543,A 0.000,B 0.000,C 90.000,E1 313.743} C_DIS
LIN {X -0.044,Y -537.872,Z 1108.540,A 0.000,B 0.000,C 90.000,E1 313.176} C_DIS
LIN {X 0.308,Y -535.165,Z 1108.536,A 0.000,B 0.000,C 90.000,E1 312.447} C_DIS
LIN {X -0.103,Y -533.653,Z 1108.533,A 0.000,B 0.000,C 90.000,E1 311.919} C_DIS
LIN {X 0.228,Y -532.391,Z 1108.530,A 0.000,B 0.000,C 90.000,E1 311.310} C_DIS
LIN {X -0.003,Y -532.230,Z 1108.529,A 0.000,B 0.000,C 90.000,E1 311.191} C_DIS
LIN {X -0.185,Y -532.218,Z 1108.528,A 0.000,B 0.000,C 90.000,E1 311.067} C_DIS
LIN {X -0.200,Y -531.863,Z 1108.526,A 0.000,B 0.000,C 90.000,E1 310.782} C_DIS
LIN {X 0.132,Y -531.313,Z 1108.525,A 0.000,B 0.000,C 90.000,E1 310.458} C_DIS
LIN {X -0.022,Y -530.748,Z 1108.521,A 0.000,B 0.000,C 90.000,E1 309.688} C_DIS
LIN {X -0.047,Y -530.463,Z 1108.517,A 0.000,B 0.000,C 90.000,E1 309.116} C_DIS
LIN {X 0.111,Y -530.357,Z 1108.516,A 0.000,B 0.000,C 90.000,E1 308.955} C_DIS
LIN {X -0.080,Y -530.407,Z 1108.514,A 0.000,B 0.000,C 90.000,E1 308.543} C_DIS
LIN {X -0.111,Y -530.304,Z 1108.511,A 0.000,B 0.000,C 90.000,E1 307.971} C_DIS
LIN {X 0.163,Y -531.783,Z 1108.492,A 0.000,B 0.000,C 90.000,E1 304.485} C_DIS
LIN {X 0.233,Y -532.777,Z 1108.482,A 0.000,B 0.000,C 90.000,E1 302.752} C_DIS
LIN {X -0.265,Y -534.305,Z 1108.471,A 0.000,B 0.000,C 90.000,E1 300.797} C_DIS
LIN {X 0.047,Y -535.117,Z 1108.465,A 0.000,B 0.000,C 90.000,E1 299.617} C_DIS
LIN {X -0.094,Y -535.902,Z 1108.458,A 0.000,B 0.000,C 90.000,E1 298.487} C_DIS
LIN {X 0.161,Y -536.767,Z 1108.449,A 0.000,B 0.000,C 90.000,E1 296.744} C_DIS
LIN {X 0.259,Y -537.250,Z 1108.442,A 0.000,B 0.000,C 90.000,E1 295.591} C_DIS
LIN {X 0.135,Y -537.612,Z 1108.436,A 0.000,B 0.000,C 90.000,E1 294.463} C_DIS
LIN {X -0.258,Y -537.912,Z 1108.428,A 0.000,B 0.000,C 90.000,E1 293.078} C_DIS
LIN {X -0.160,Y -538.096,Z 1108.420,A 0.000,B 0.000,C 90.000,E1 291.642} C_DIS
LIN {X 0.019,Y -538.193,Z 1108.414,A 0.000,B 0.000,C 90.000,E1 290.482} C_DIS
LIN {X -0.268,Y -538.037,Z 1108.406,A 0.000,B 0.000,C 90.000,E1 289.087} C_DIS
LIN {X 0.164,Y -537.694,Z 1108.396,A 0.000,B 0.000,C 90.000,E1 287.330} C_DIS
LIN {X 0.213,Y -537.293,Z 1108.389,A 0.000,B 0.000,C 90.000,E1 285.898} C_DIS
LIN {X 0.117,Y -536.721,Z 1108.381,A 0.000,B 0.000,C 90.000,E1 284.481} C_DIS
LIN {X 0.131,Y -535.759,Z 1108.370,A 0.000,B 0.000,C 90.000,E1 282.479} C_DIS
LIN {X -0.106,Y -535.061,Z 1108.361,A 0.000,B 0.000,C 90.000,E1 281.074} C_DIS
LIN {X 0.264,Y -534.055,Z 1108.350,A 0.000,B 0.000,C 90.000,E1 279.029} C_DIS
LIN {X -0.171,Y -533.088,Z 1108.339,A 0.000,B 0.000,C 90.000,E1 277.068} C_DIS
LIN {X -0.090,Y -532.102,Z 1108.328,A 0.000,B 0.000,C 90.000,E1 275.049} C_DIS
LIN {X -0.096,Y -531.190,Z 1108.317,A 0.000,B 0.000,C 90.000,E1 273.037} C_DIS
LIN {X -0.187,Y -530.262,Z 1108.306,A 0.000,B 0.000,C 90.000,E1 271.031} C_DIS
LIN {X 0.242,Y -529.451,Z 1108.296,A 0.000,B 0.000,C 90.000,E1 269.255} C_DIS
LIN {X 0.156,Y -528.717,Z 1108.288,A 0.000,B 0.000,C 90.000,E1 267.822} C_DIS
LIN {X 0.028,Y -527.650,Z 1108.278,A 0.000,B 0.000,C 90.000,E1 266.102} C_DIS
LIN {X -0.062,Y -526.779,Z 1108.270,A 0.000,B 0.000,C 90.000,E1 264.666} C_DIS
LIN {X -0.128,Y -525.874,Z 1108.264,A 0.000,B 0.000,C 90.000,E1 263.514} C_DIS
LIN {X -0.144,Y -524.746,Z 1108.257,A 0.000,B 0.000,C 90.000,E1 262.356} C_DIS
LIN {X -0.214,Y -522.397,Z 1108.245,A 0.000,B 0.000,C 90.000,E1 260.038} C_DIS
LIN {X -0.185,Y -521.305,Z 1108.238,A 0.000,B 0.000,C 90.000,E1 258.870} C_DIS
LIN {X -0.171,Y -519.639,Z 1108.228,A 0.000,B 0.000,C 90.000,E1 257.117} C_DIS
LIN {X 0.040,Y -518.001,Z 1108.219,A 0.000,B 0.000,C 90.000,E1 255.338} C_DIS
LIN {X 0.096,Y -516.432,Z 1108.210,A 0.000,B 0.000,C 90.000,E1 253.866} C_DIS
LIN {X -0.122,Y -514.606,Z 1108.201,A 0.000,B 0.000,C 90.000,E1 252.127} C_DIS
LIN {X -0.217,Y -512.761,Z 1108.191,A 0.000,B 0.000,C 90.000,E1 250.369} C_DIS
LIN {X -0.066,Y -510.308,Z 1108.179,A 0.000,B 0.000,C 90.000,E1 248.284} C_DIS
LIN {X -0.101,Y -508.927,Z 1108.173,A 0.000,B 0.000,C 90.000,E1 247.102} C_DIS
LIN {X -0.158,Y -507.246,Z 1108.166,A 0.000,B 0.000,C 90.000,E1 245.921} C_DIS
LIN {X -0.032,Y -505.556,Z 1108.160,A 0.000,B 0.000,C 90.000,E1 244.717} C_DIS
LIN {X 0.143,Y -503.154,Z 1108.151,A 0.000,B 0.000,C 90.000,E1 243.204} C_DIS
LIN {X -0.104,Y -500.261,Z 1108.141,A 0.000,B 0.000,C 90.000,E1 241.435} C_DIS
LIN {X 0.158,Y -496.252,Z 1108.128,A 0.000,B 0.000,C 90.000,E1 238.997} C_DIS
LIN {X 0.154,Y -494.144,Z 1108.121,A 0.000,B 0.000,C 90.000,E1 237.788} C_DIS
LIN {X -0.196,Y -490.967,Z 1108.111,A 0.000,B 0.000,C 90.000,E1 236.008} C_DIS
LIN {X -0.017,Y -488.751,Z 1108.104,A 0.000,B 0.000,C 90.000,E1 234.769} C_DIS
LIN {X -0.154,Y -485.899,Z 1108.096,A 0.000,B 0.000,C 90.000,E1 233.256} C_DIS
LIN {X 0.222,Y -483.567,Z 1108.089,A 0.000,B 0.000,C 90.000,E1 231.984} C_DIS
LIN {X -0.086,Y -480.534,Z 1108.080,A 0.000,B 0.000,C 90.000,E1 230.481} C_DIS
LIN {X 0.032,Y -476.894,Z 1108.070,A 0.000,B 0.000,C 90.000,E1 228.609} C_DIS
LIN {X -0.206,Y -472.729,Z 1108.058,A 0.000,B 0.000,C 90.000,E1 226.458} C_DIS
LIN {X 0.002,Y -469.300,Z 1108.048,A 0.000,B 0.000,C 90.000,E1 224.555} C_DIS
LIN {X 0.058,Y -466.495,Z 1108.039,A 0.000,B 0.000,C 90.000,E1 222.975} C_DIS
LIN {X 0.149,Y -463.180,Z 1108.028,A 0.000,B 0.000,C 90.000,E1 221.067} C_DIS
LIN {X 0.258,Y -459.585,Z 1108.016,A 0.000,B 0.000,C 90.000,E1 218.830} C_DIS
LIN {X -0.031,Y -456.598,Z 1108.005,A 0.000,B 0.000,C 90.000,E1 216.950} C_DIS
LIN {X -0.024,Y -453.727,Z 1107.995,A 0.000,B 0.000,C 90.000,E1 215.025} C_DIS
LIN {X 0.023,Y -450.886,Z 1107.984,A 0.000,B 0.000,C 90.000,E1 213.086} C_DIS
LIN {X 0.136,Y -448.215,Z 1107.973,A 0.000,B 0.000,C 90.000,E1 211.131} C_DIS
LIN {X -0.068,Y -444.601,Z 1107.957,A 0.000,B 0.000,C 90.000,E1 208.231} C_DIS
LIN {X 0.018,Y -441.665,Z 1107.939,A 0.000,B 0.000,C 90.000,E1 204.951} C_DIS
LIN {X 0.149,Y -441.290,Z 1107.933,A 0.000,B 0.000,C 90.000,E1 203.951} C_DIS
LIN {X 0.127,Y -441.507,Z 1107.926,A 0.000,B 0.000,C 90.000,E1 202.642} C_DIS
LIN {X 0.091,Y -442.214,Z 1107.920,A 0.000,B 0.000,C 90.000,E1 201.663} C_DIS
LIN {X -0.201,Y -442.896,Z 1107.917,A 0.000,B 0.000,C 90.000,E1 201.046} C_DIS
LIN {X -0.218,Y -444.680,Z 1107.911,A 0.000,B 0.000,C 90.000,E1 200.066} C_DIS
LIN {X -0.216,Y -446.987,Z 1107.906,A 0.000,B 0.000,C 90.000,E1 199.087} C_DIS
LIN {X 0.234,Y -449.719,Z 1107.901,A 0.000,B 0.000,C 90.000,E1 198.055} C_DIS
LIN {X -0.140,Y -457.452,Z 1107.888,A 0.000,B 0.000,C 90.000,E1 195.843} C_DIS
LIN {X -0.160,Y -467.528,Z 1107.874,A 0.000,B 0.000,C 90.000,E1 193.300} C_DIS
LIN {X -0.221,Y -479.639,Z 1107.858,A 0.000,B 0.000,C 90.000,E1 190.489} C_DIS
LIN {X 0.165,Y -485.172,Z 1107.851,A 0.000,B 0.000,C 90.000,E1 189.208} C_DIS
LIN {X -0.187,Y -491.391,Z 1107.844,A 0.000,B 0.000,C 90.000,E1 187.871} C_DIS
LIN {X -0.023,Y -497.515,Z 1107.836,A 0.000,B 0.000,C 90.000,E1 186.486} C_DIS
LIN {X 0.076,Y -504.706,Z 1107.827,A 0.000,B 0.000,C 90.000,E1 184.821} C_DIS
LIN {X 0.069,Y -512.687,Z 1107.817,A 0.000,B 0.000,C 90.000,E1 183.037} C_DIS
LIN {X -0.115,Y -521.210,Z 1107.806,A 0.000,B 0.000,C 90.000,E1 181.146} C_DIS
LIN {X 0.234,Y -526.568,Z 1107.800,A 0.000,B 0.000,C 90.000,E1 179.943} C_DIS
LIN {X -0.149,Y -533.823,Z 1107.791,A 0.000,B 0.000,C 90.000,E1 178.396} C_DIS
LIN {X -0.123,Y -540.386,Z 1107.783,A 0.000,B 0.000,C 90.000,E1 176.963} C_DIS
LIN {X 0.056,Y -546.877,Z 1107.775,A 0.000,B 0.000,C 90.000,E1 175.527} C_DIS
LIN {X 0.166,Y -553.930,Z 1107.767,A 0.000,B 0.000,C 90.000,E1 173.970} C_DIS
LIN {X -0.132,Y -561.066,Z 1107.758,A 0.000,B 0.000,C 90.000,E1 172.470} C_DIS
LIN {X -0.236,Y -566.153,Z 1107.752,A 0.000,B 0.000,C 90.000,E1 171.376} C_DIS
LIN {X -0.143,Y -572.976,Z 1107.744,A 0.000,B 0.000,C 90.000,E1 169.859} C_DIS
LIN {X 0.214,Y -579.050,Z 1107.736,A 0.000,B 0.000,C 90.000,E1 168.465} C_DIS
LIN {X -0.254,Y -582.555,Z 1107.732,A 0.000,B 0.000,C 90.000,E1 167.701} C_DIS
LIN {X 0.123,Y -587.086,Z 1107.726,A 0.000,B 0.000,C 90.000,E1 166.589} C_DIS
LIN {X 0.133,Y -591.385,Z 1107.720,A 0.000,B 0.000,C 90.000,E1 165.519} C_DIS
LIN {X 0.209,Y -595.458,Z 1107.714,A 0.000,B 0.000,C 90.000,E1 164.448} C_DIS
LIN {X 0.343,Y -599.326,Z 1107.708,A 0.000,B 0.000,C 90.000,E1 163.378} C_DIS
LIN {X 0.233,Y -602.052,Z 1107.703,A 0.000,B 0.000,C 90.000,E1 162.598} C_DIS
LIN {X -0.130,Y -605.509,Z 1107.698,A 0.000,B 0.000,C 90.000,E1 161.583} C_DIS
LIN {X -0.261,Y -608.757,Z 1107.692,A 0.000,B 0.000,C 90.000,E1 160.550} C_DIS
LIN {X 0.174,Y -612.611,Z 1107.685,A 0.000,B 0.000,C 90.000,E1 159.209} C_DIS
LIN {X 0.098,Y -616.204,Z 1107.677,A 0.000,B 0.000,C 90.000,E1 157.922} C_DIS
LIN {X -0.254,Y -619.688,Z 1107.670,A 0.000,B 0.000,C 90.000,E1 156.666} C_DIS
LIN {X 0.026,Y -623.049,Z 1107.663,A 0.000,B 0.000,C 90.000,E1 155.357} C_DIS
LIN {X 0.058,Y -626.273,Z 1107.656,A 0.000,B 0.000,C 90.000,E1 154.076} C_DIS
LIN {X 0.152,Y -629.331,Z 1107.649,A 0.000,B 0.000,C 90.000,E1 152.794} C_DIS
LIN {X -0.200,Y -633.258,Z 1107.639,A 0.000,B 0.000,C 90.000,E1 151.051} C_DIS
LIN {X -0.252,Y -636.004,Z 1107.632,A 0.000,B 0.000,C 90.000,E1 149.793} C_DIS
LIN {X -0.259,Y -638.600,Z 1107.625,A 0.000,B 0.000,C 90.000,E1 148.535} C_DIS
LIN {X 0.107,Y -641.091,Z 1107.618,A 0.000,B 0.000,C 90.000,E1 147.248} C_DIS
LIN {X -0.022,Y -643.490,Z 1107.611,A 0.000,B 0.000,C 90.000,E1 146.008} C_DIS
LIN {X -0.115,Y -645.736,Z 1107.604,A 0.000,B 0.000,C 90.000,E1 144.769} C_DIS
LIN {X 0.150,Y -648.824,Z 1107.595,A 0.000,B 0.000,C 90.000,E1 143.004} C_DIS
LIN {X -0.146,Y -651.931,Z 1107.585,A 0.000,B 0.000,C 90.000,E1 141.295} C_DIS
LIN {X 0.143,Y -655.167,Z 1107.575,A 0.000,B 0.000,C 90.000,E1 139.542} C_DIS
LIN {X -0.036,Y -657.993,Z 1107.567,A 0.000,B 0.000,C 90.000,E1 138.081} C_DIS
LIN {X -0.138,Y -660.475,Z 1107.560,A 0.000,B 0.000,C 90.000,E1 136.863} C_DIS
LIN {X -0.270,Y -665.233,Z 1107.548,A 0.000,B 0.000,C 90.000,E1 134.676} C_DIS
LIN {X 0.217,Y -669.814,Z 1107.537,A 0.000,B 0.000,C 90.000,E1 132.690} C_DIS
LIN {X 0.347,Y -674.033,Z 1107.528,A 0.000,B 0.000,C 90.000,E1 130.987} C_DIS
LIN {X 0.098,Y -677.577,Z 1107.520,A 0.000,B 0.000,C 90.000,E1 129.564} C_DIS
LIN {X 0.049,Y -681.899,Z 1107.511,A 0.000,B 0.000,C 90.000,E1 127.890} C_DIS
LIN {X -0.102,Y -684.947,Z 1107.504,A 0.000,B 0.000,C 90.000,E1 126.710} C_DIS
LIN {X 0.120,Y -688.518,Z 1107.496,A 0.000,B 0.000,C 90.000,E1 125.264} C_DIS
LIN {X -0.137,Y -691.988,Z 1107.488,A 0.000,B 0.000,C 90.000,E1 123.865} C_DIS
LIN {X 0.005,Y -694.888,Z 1107.482,A 0.000,B 0.000,C 90.000,E1 122.673} C_DIS
LIN {X 0.152,Y -697.114,Z 1107.476,A 0.000,B 0.000,C 90.000,E1 121.720} C_DIS
LIN {X 0.307,Y -698.625,Z 1107.472,A 0.000,B 0.000,C 90.000,E1 121.003} C_DIS
LIN {X 0.146,Y -700.390,Z 1107.467,A 0.000,B 0.000,C 90.000,E1 120.079} C_DIS
LIN {X 0.008,Y -701.952,Z 1107.462,A 0.000,B 0.000,C 90.000,E1 119.155} C_DIS
LIN {X -0.114,Y -703.329,Z 1107.457,A 0.000,B 0.000,C 90.000,E1 118.231} C_DIS
LIN {X 0.110,Y -704.211,Z 1107.453,A 0.000,B 0.000,C 90.000,E1 117.513} C_DIS
LIN {X 0.023,Y -704.807,Z 1107.449,A 0.000,B 0.000,C 90.000,E1 116.821} C_DIS
LIN {X -0.104,Y -705.646,Z 1107.443,A 0.000,B 0.000,C 90.000,E1 115.668} C_DIS
LIN {X -0.160,Y -705.866,Z 1107.440,A 0.000,B 0.000,C 90.000,E1 115.207} C_DIS
LIN {X 0.124,Y -705.814,Z 1107.437,A 0.000,B 0.000,C 90.000,E1 114.719} C_DIS
LIN {X -0.226,Y -705.673,Z 1107.436,A 0.000,B 0.000,C 90.000,E1 114.515} C_DIS
LIN {X 0.063,Y -704.934,Z 1107.434,A 0.000,B 0.000,C 90.000,E1 114.027} C_DIS
LIN {X -0.294,Y -704.208,Z 1107.432,A 0.000,B 0.000,C 90.000,E1 113.823} C_DIS
LIN {X -0.009,Y -702.307,Z 1107.430,A 0.000,B 0.000,C 90.000,E1 113.334} C_DIS
LIN {X 0.130,Y -701.533,Z 1107.429,A 0.000,B 0.000,C 90.000,E1 113.206} C_DIS
LIN {X -0.248,Y -697.393,Z 1107.426,A 0.000,B 0.000,C 90.000,E1 112.770} C_DIS
LIN {X -0.117,Y -696.018,Z 1107.426,A 0.000,B 0.000,C 90.000,E1 112.642} C_DIS
LIN {X 0.110,Y -693.959,Z 1107.425,A 0.000,B 0.000,C 90.000,E1 112.514} C_DIS
LIN {X 0.089,Y -686.297,Z 1107.423,A 0.000,B 0.000,C 90.000,E1 112.206} C_DIS
LIN {X -0.082,Y -682.706,Z 1107.423,A 0.000,B 0.000,C 90.000,E1 112.153} C_DIS
LIN {X -0.053,Y -676.063,Z 1107.423,A 0.000,B 0.000,C 90.000,E1 112.078} C_DIS
LIN {X -0.097,Y -603.938,Z 1107.423,A 0.000,B 0.000,C 90.000,E1 112.078} C_DIS
LIN {X 0.218,Y -600.318,Z 1107.422,A 0.000,B 0.000,C 90.000,E1 111.844} C_DIS
LIN {X 0.044,Y -595.777,Z 1107.420,A 0.000,B 0.000,C 90.000,E1 111.535} C_DIS
LIN {X 0.069,Y -578.760,Z 1107.412,A 0.000,B 0.000,C 90.000,E1 110.066} C_DIS
LIN {X 0.112,Y -574.531,Z 1107.410,A 0.000,B 0.000,C 90.000,E1 109.704} C_DIS
LIN {X -0.068,Y -568.453,Z 1107.407,A 0.000,B 0.000,C 90.000,E1 109.268} C_DIS
LIN {X 0.200,Y -560.171,Z 1107.404,A 0.000,B 0.000,C 90.000,E1 108.725} C_DIS
LIN {X 0.162,Y -553.946,Z 1107.402,A 0.000,B 0.000,C 90.000,E1 108.362} C_DIS
LIN {X 0.173,Y -549.897,Z 1107.401,A 0.000,B 0.000,C 90.000,E1 108.055} C_DIS
LIN {X 0.144,Y -548.647,Z 1107.399,A 0.000,B 0.000,C 90.000,E1 107.873} C_DIS
LIN {X 0.102,Y -548.620,Z 1107.399,A 0.000,B 0.000,C 90.000,E1 107.873} C_DIS
LIN {X 0.267,Y -548.296,Z 1107.397,A 0.000,B 0.000,C 90.000,E1 107.457} C_DIS
LIN {X -0.083,Y -548.605,Z 1107.393,A 0.000,B 0.000,C 90.000,E1 106.732} C_DIS
LIN {X 0.025,Y -549.597,Z 1107.385,A 0.000,B 0.000,C 90.000,E1 105.315} C_DIS
LIN {X 0.097,Y -551.307,Z 1107.373,A 0.000,B 0.000,C 90.000,E1 103.063} C_DIS
LIN {X -0.038,Y -553.310,Z 1107.360,A 0.000,B 0.000,C 90.000,E1 100.838} C_DIS
LIN {X 0.195,Y -555.256,Z 1107.349,A 0.000,B 0.000,C 90.000,E1 98.859} C_DIS
LIN {X 0.128,Y -556.695,Z 1107.342,A 0.000,B 0.000,C 90.000,E1 97.473} C_DIS
LIN {X 0.023,Y -557.836,Z 1107.335,A 0.000,B 0.000,C 90.000,E1 96.372} C_DIS
LIN {X -0.137,Y -558.938,Z 1107.329,A 0.000,B 0.000,C 90.000,E1 95.277} C_DIS
LIN {X -0.203,Y -560.092,Z 1107.322,A 0.000,B 0.000,C 90.000,E1 93.898} C_DIS
LIN {X 0.183,Y -560.858,Z 1107.315,A 0.000,B 0.000,C 90.000,E1 92.751} C_DIS
LIN {X -0.094,Y -561.381,Z 1107.311,A 0.000,B 0.000,C 90.000,E1 91.949} C_DIS
LIN {X -0.050,Y -562.314,Z 1107.302,A 0.000,B 0.000,C 90.000,E1 90.286} C_DIS
LIN {X -0.001,Y -563.094,Z 1107.292,A 0.000,B 0.000,C 90.000,E1 88.625} C_DIS
LIN {X -0.029,Y -563.785,Z 1107.285,A 0.000,B 0.000,C 90.000,E1 87.249} C_DIS
LIN {X 0.092,Y -564.514,Z 1107.276,A 0.000,B 0.000,C 90.000,E1 85.584} C_DIS
LIN {X 0.281,Y -565.186,Z 1107.266,A 0.000,B 0.000,C 90.000,E1 83.913} C_DIS
LIN {X 0.085,Y -565.892,Z 1107.256,A 0.000,B 0.000,C 90.000,E1 82.008} C_DIS
LIN {X -0.192,Y -566.452,Z 1107.247,A 0.000,B 0.000,C 90.000,E1 80.387} C_DIS
LIN {X -0.194,Y -567.286,Z 1107.236,A 0.000,B 0.000,C 90.000,E1 78.465} C_DIS
LIN {X 0.060,Y -568.232,Z 1107.225,A 0.000,B 0.000,C 90.000,E1 76.520} C_DIS
LIN {X -0.029,Y -569.450,Z 1107.213,A 0.000,B 0.000,C 90.000,E1 74.338} C_DIS
LIN {X 0.211,Y -571.063,Z 1107.201,A 0.000,B 0.000,C 90.000,E1 72.127} C_DIS
LIN {X 0.140,Y -572.321,Z 1107.192,A 0.000,B 0.000,C 90.000,E1 70.496} C_DIS
LIN {X -0.249,Y -573.827,Z 1107.183,A 0.000,B 0.000,C 90.000,E1 68.901} C_DIS
LIN {X -0.017,Y -575.523,Z 1107.172,A 0.000,B 0.000,C 90.000,E1 66.975} C_DIS
LIN {X -0.121,Y -576.867,Z 1107.163,A 0.000,B 0.000,C 90.000,E1 65.357} C_DIS
LIN {X -0.194,Y -577.718,Z 1107.157,A 0.000,B 0.000,C 90.000,E1 64.280} C_DIS
LIN {X -0.142,Y -578.706,Z 1107.150,A 0.000,B 0.000,C 90.000,E1 62.922} C_DIS
LIN {X -0.198,Y -579.519,Z 1107.144,A 0.000,B 0.000,C 90.000,E1 61.847} C_DIS
LIN {X 0.018,Y -580.536,Z 1107.135,A 0.000,B 0.000,C 90.000,E1 60.205} C_DIS
LIN {X -0.104,Y -581.325,Z 1107.127,A 0.000,B 0.000,C 90.000,E1 58.869} C_DIS
LIN {X -0.069,Y -581.977,Z 1107.121,A 0.000,B 0.000,C 90.000,E1 57.788} C_DIS
LIN {X 0.343,Y -583.074,Z 1107.109,A 0.000,B 0.000,C 90.000,E1 55.595} C_DIS
LIN {X 0.269,Y -583.787,Z 1107.100,A 0.000,B 0.000,C 90.000,E1 53.989} C_DIS
LIN {X 0.181,Y -584.187,Z 1107.094,A 0.000,B 0.000,C 90.000,E1 52.924} C_DIS
LIN {X -0.368,Y -584.589,Z 1107.088,A 0.000,B 0.000,C 90.000,E1 51.904} C_DIS
LIN {X -0.271,Y -584.748,Z 1107.084,A 0.000,B 0.000,C 90.000,E1 51.090} C_DIS
LIN {X -0.173,Y -584.807,Z 1107.079,A 0.000,B 0.000,C 90.000,E1 50.275} C_DIS
LIN {X -0.160,Y -584.669,Z 1107.072,A 0.000,B 0.000,C 90.000,E1 48.933} C_DIS
LIN {X 0.059,Y -584.464,Z 1107.066,A 0.000,B 0.000,C 90.000,E1 47.838} C_DIS
LIN {X 0.020,Y -584.051,Z 1107.058,A 0.000,B 0.000,C 90.000,E1 46.500} C_DIS
LIN {X -0.029,Y -583.380,Z 1107.051,A 0.000,B 0.000,C 90.000,E1 45.162} C_DIS
LIN {X -0.248,Y -582.708,Z 1107.045,A 0.000,B 0.000,C 90.000,E1 44.109} C_DIS
LIN {X -0.058,Y -581.717,Z 1107.039,A 0.000,B 0.000,C 90.000,E1 43.014} C_DIS
LIN {X -0.040,Y -580.877,Z 1107.035,A 0.000,B 0.000,C 90.000,E1 42.204} C_DIS
LIN {X -0.108,Y -579.119,Z 1107.027,A 0.000,B 0.000,C 90.000,E1 40.862} C_DIS
LIN {X 0.306,Y -577.998,Z 1107.022,A 0.000,B 0.000,C 90.000,E1 40.011} C_DIS
LIN {X 0.037,Y -576.143,Z 1107.016,A 0.000,B 0.000,C 90.000,E1 38.955} C_DIS
LIN {X -0.168,Y -574.035,Z 1107.010,A 0.000,B 0.000,C 90.000,E1 37.890} C_DIS
LIN {X -0.186,Y -572.162,Z 1107.006,A 0.000,B 0.000,C 90.000,E1 37.076} C_DIS
LIN {X 0.227,Y -570.053,Z 1107.001,A 0.000,B 0.000,C 90.000,E1 36.217} C_DIS
LIN {X -0.181,Y -567.601,Z 1106.997,A 0.000,B 0.000,C 90.000,E1 35.438} C_DIS
LIN {X -0.037,Y -563.747,Z 1106.991,A 0.000,B 0.000,C 90.000,E1 34.326} C_DIS
LIN {X -0.141,Y -561.555,Z 1106.988,A 0.000,B 0.000,C 90.000,E1 33.785} C_DIS
LIN {X 0.026,Y -557.327,Z 1106.982,A 0.000,B 0.000,C 90.000,E1 32.801} C_DIS
LIN {X -0.238,Y -554.052,Z 1106.978,A 0.000,B 0.000,C 90.000,E1 32.133} C_DIS
LIN {X -0.009,Y -549.054,Z 1106.973,A 0.000,B 0.000,C 90.000,E1 31.131} C_DIS
LIN {X 0.281,Y -544.336,Z 1106.968,A 0.000,B 0.000,C 90.000,E1 30.256} C_DIS
LIN {X 0.245,Y -539.429,Z 1106.964,A 0.000,B 0.000,C 90.000,E1 29.411} C_DIS
LIN {X -0.169,Y -534.895,Z 1106.960,A 0.000,B 0.000,C 90.000,E1 28.743} C_DIS
LIN {X -0.156,Y -529.920,Z 1106.956,A 0.000,B 0.000,C 90.000,E1 28.025} C_DIS
LIN {X 0.300,Y -524.574,Z 1106.952,A 0.000,B 0.000,C 90.000,E1 27.257} C_DIS
LIN {X 0.140,Y -520.009,Z 1106.948,A 0.000,B 0.000,C 90.000,E1 26.693} C_DIS
LIN {X 0.132,Y -513.839,Z 1106.944,A 0.000,B 0.000,C 90.000,E1 25.976} C_DIS
LIN {X -0.188,Y -507.279,Z 1106.940,A 0.000,B 0.000,C 90.000,E1 25.283} C_DIS
LIN {X 0.026,Y -496.465,Z 1106.934,A 0.000,B 0.000,C 90.000,E1 24.131} C_DIS
LIN {X 0.161,Y -485.208,Z 1106.928,A 0.000,B 0.000,C 90.000,E1 23.025} C_DIS
LIN {X -0.151,Y -477.907,Z 1106.924,A 0.000,B 0.000,C 90.000,E1 22.386} C_DIS
LIN {X -0.053,Y -467.517,Z 1106.919,A 0.000,B 0.000,C 90.000,E1 21.461} C_DIS
LIN {X 0.275,Y -451.326,Z 1106.911,A 0.000,B 0.000,C 90.000,E1 19.993} C_DIS
LIN {X 0.161,Y -432.415,Z 1106.901,A 0.000,B 0.000,C 90.000,E1 18.236} C_DIS
LIN {X -0.097,Y -418.514,Z 1106.893,A 0.000,B 0.000,C 90.000,E1 16.804} C_DIS
LIN {X 0.035,Y -408.949,Z 1106.887,A 0.000,B 0.000,C 90.000,E1 15.662} C_DIS
LIN {X 0.072,Y -399.949,Z 1106.881,A 0.000,B 0.000,C 90.000,E1 14.481} C_DIS
LIN {X -0.101,Y -396.785,Z 1106.878,A 0.000,B 0.000,C 90.000,E1 14.008} C_DIS
LIN {X -0.065,Y -395.823,Z 1106.877,A 0.000,B 0.000,C 90.000,E1 13.828} C_DIS
LIN {X 0.016,Y -393.835,Z 1106.874,A 0.000,B 0.000,C 90.000,E1 13.355} C_DIS
LIN {X 0.138,Y -393.311,Z 1106.873,A 0.000,B 0.000,C 90.000,E1 13.175} C_DIS
LIN {X -0.010,Y -392.175,Z 1106.870,A 0.000,B 0.000,C 90.000,E1 12.591} C_DIS
LIN {X 0.123,Y -392.067,Z 1106.867,A 0.000,B 0.000,C 90.000,E1 11.951} C_DIS
LIN {X -0.075,Y -392.614,Z 1106.863,A 0.000,B 0.000,C 90.000,E1 11.422} C_DIS
LIN {X 0.182,Y -395.695,Z 1106.854,A 0.000,B 0.000,C 90.000,E1 9.613} C_DIS
LIN {X 0.065,Y -398.822,Z 1106.846,A 0.000,B 0.000,C 90.000,E1 8.219} C_DIS
LIN {X -0.059,Y -402.310,Z 1106.838,A 0.000,B 0.000,C 90.000,E1 6.834} C_DIS
LIN {X -0.128,Y -404.866,Z 1106.832,A 0.000,B 0.000,C 90.000,E1 5.796} C_DIS
LIN {X -0.152,Y -406.393,Z 1106.829,A 0.000,B 0.000,C 90.000,E1 5.277} C_DIS
LIN {X -0.171,Y -407.046,Z 1106.828,A 0.000,B 0.000,C 90.000,E1 5.106} C_DIS
LIN {X -0.152,Y -410.706,Z 1106.824,A 0.000,B 0.000,C 90.000,E1 4.416} C_DIS
LIN {X -0.162,Y -411.902,Z 1106.823,A 0.000,B 0.000,C 90.000,E1 4.245} C_DIS
LIN {X 0.142,Y -416.953,Z 1106.821,A 0.000,B 0.000,C 90.000,E1 3.726} C_DIS
LIN {X 0.006,Y -432.199,Z 1106.815,A 0.000,B 0.000,C 90.000,E1 2.694} C_DIS
LIN {X -0.001,Y -450.306,Z 1106.808,A 0.000,B 0.000,C 90.000,E1 1.489} C_DIS
LIN {X 0.213,Y -465.067,Z 1106.803,A 0.000,B 0.000,C 90.000,E1 0.516} C_DIS
LIN {X -0.189,Y -478.451,Z 1106.798,A 0.000,B 0.000,C 90.000,E1 359.714} C_DIS
LIN {X -0.146,Y -487.990,Z 1106.795,A 0.000,B 0.000,C 90.000,E1 359.083} C_DIS
LIN {X 0.158,Y -495.744,Z 1106.792,A 0.000,B 0.000,C 90.000,E1 358.511} C_DIS
LIN {X -0.129,Y -503.246,Z 1106.789,A 0.000,B 0.000,C 90.000,E1 357.993} C_DIS
LIN {X 0.252,Y -510.650,Z 1106.786,A 0.000,B 0.000,C 90.000,E1 357.364} C_DIS
LIN {X 0.057,Y -516.441,Z 1106.783,A 0.000,B 0.000,C 90.000,E1 356.906} C_DIS
LIN {X 0.051,Y -523.286,Z 1106.779,A 0.000,B 0.000,C 90.000,E1 356.274} C_DIS
LIN {X 0.202,Y -529.946,Z 1106.776,A 0.000,B 0.000,C 90.000,E1 355.584} C_DIS
LIN {X 0.081,Y -536.182,Z 1106.772,A 0.000,B 0.000,C 90.000,E1 354.894} C_DIS
LIN {X 0.249,Y -540.679,Z 1106.769,A 0.000,B 0.000,C 90.000,E1 354.318} C_DIS
LIN {X 0.144,Y -545.796,Z 1106.765,A 0.000,B 0.000,C 90.000,E1 353.628} C_DIS
LIN {X 0.063,Y -550.502,Z 1106.761,A 0.000,B 0.000,C 90.000,E1 352.932} C_DIS
LIN {X 0.206,Y -553.981,Z 1106.758,A 0.000,B 0.000,C 90.000,E1 352.356} C_DIS
LIN {X 0.201,Y -557.762,Z 1106.754,A 0.000,B 0.000,C 90.000,E1 351.659} C_DIS
LIN {X -0.159,Y -560.499,Z 1106.751,A 0.000,B 0.000,C 90.000,E1 351.141} C_DIS
LIN {X 0.140,Y -563.067,Z 1106.748,A 0.000,B 0.000,C 90.000,E1 350.557} C_DIS
LIN {X -0.030,Y -566.540,Z 1106.743,A 0.000,B 0.000,C 90.000,E1 349.746} C_DIS
LIN {X 0.119,Y -570.817,Z 1106.737,A 0.000,B 0.000,C 90.000,E1 348.634} C_DIS
LIN {X 0.012,Y -573.826,Z 1106.732,A 0.000,B 0.000,C 90.000,E1 347.825} C_DIS
LIN {X 0.180,Y -576.613,Z 1106.728,A 0.000,B 0.000,C 90.000,E1 346.992} C_DIS
LIN {X 0.125,Y -580.864,Z 1106.720,A 0.000,B 0.000,C 90.000,E1 345.644} C_DIS
LIN {X 0.049,Y -584.086,Z 1106.714,A 0.000,B 0.000,C 90.000,E1 344.574} C_DIS
LIN {X -0.309,Y -587.999,Z 1106.707,A 0.000,B 0.000,C 90.000,E1 343.268} C_DIS
LIN {X -0.119,Y -590.943,Z 1106.701,A 0.000,B 0.000,C 90.000,E1 342.181} C_DIS
LIN {X 0.118,Y -593.749,Z 1106.695,A 0.000,B 0.000,C 90.000,E1 341.094} C_DIS
LIN {X 0.289,Y -596.898,Z 1106.688,A 0.000,B 0.000,C 90.000,E1 339.752} C_DIS
LIN {X 0.043,Y -599.167,Z 1106.682,A 0.000,B 0.000,C 90.000,E1 338.720} C_DIS
LIN {X -0.130,Y -600.209,Z 1106.679,A 0.000,B 0.000,C 90.000,E1 338.209} C_DIS
LIN {X 0.136,Y -602.364,Z 1106.672,A 0.000,B 0.000,C 90.000,E1 336.869} C_DIS
LIN {X -0.070,Y -603.444,Z 1106.667,A 0.000,B 0.000,C 90.000,E1 336.102} C_DIS
LIN {X -0.020,Y -604.703,Z 1106.661,A 0.000,B 0.000,C 90.000,E1 335.049} C_DIS
LIN {X -0.250,Y -605.744,Z 1106.656,A 0.000,B 0.000,C 90.000,E1 334.024} C_DIS
LIN {X 0.130,Y -606.277,Z 1106.651,A 0.000,B 0.000,C 90.000,E1 333.204} C_DIS
LIN {X 0.200,Y -606.745,Z 1106.646,A 0.000,B 0.000,C 90.000,E1 332.153} C_DIS
LIN {X -0.006,Y -606.832,Z 1106.640,A 0.000,B 0.000,C 90.000,E1 331.129} C_DIS
LIN {X 0.130,Y -606.439,Z 1106.635,A 0.000,B 0.000,C 90.000,E1 330.333} C_DIS
LIN {X 0.321,Y -606.127,Z 1106.632,A 0.000,B 0.000,C 90.000,E1 329.793} C_DIS
LIN {X -0.376,Y -605.211,Z 1106.628,A 0.000,B 0.000,C 90.000,E1 329.076} C_DIS
LIN {X -0.126,Y -604.861,Z 1106.627,A 0.000,B 0.000,C 90.000,E1 328.791} C_DIS
LIN {X -0.082,Y -602.976,Z 1106.621,A 0.000,B 0.000,C 90.000,E1 327.740} C_DIS
LIN {X -0.173,Y -601.200,Z 1106.616,A 0.000,B 0.000,C 90.000,E1 326.962} C_DIS
LIN {X -0.105,Y -599.217,Z 1106.612,A 0.000,B 0.000,C 90.000,E1 326.167} C_DIS
LIN {X -0.225,Y -596.959,Z 1106.608,A 0.000,B 0.000,C 90.000,E1 325.388} C_DIS
LIN {X 0.124,Y -594.554,Z 1106.603,A 0.000,B 0.000,C 90.000,E1 324.562} C_DIS
LIN {X -0.024,Y -588.667,Z 1106.593,A 0.000,B 0.000,C 90.000,E1 322.718} C_DIS
LIN {X 0.301,Y -585.050,Z 1106.587,A 0.000,B 0.000,C 90.000,E1 321.618} C_DIS
LIN {X 0.301,Y -580.636,Z 1106.579,A 0.000,B 0.000,C 90.000,E1 320.275} C_DIS
LIN {X 0.220,Y -575.462,Z 1106.572,A 0.000,B 0.000,C 90.000,E1 318.933} C_DIS
LIN {X -0.216,Y -572.053,Z 1106.568,A 0.000,B 0.000,C 90.000,E1 318.162} C_DIS
LIN {X 0.168,Y -570.300,Z 1106.565,A 0.000,B 0.000,C 90.000,E1 317.715} C_DIS
LIN {X 0.059,Y -565.936,Z 1106.561,A 0.000,B 0.000,C 90.000,E1 316.905} C_DIS
LIN {X -0.240,Y -560.481,Z 1106.555,A 0.000,B 0.000,C 90.000,E1 315.972} C_DIS
LIN {X 0.218,Y -552.135,Z 1106.548,A 0.000,B 0.000,C 90.000,E1 314.676} C_DIS
LIN {X -0.045,Y -544.937,Z 1106.542,A 0.000,B 0.000,C 90.000,E1 313.581} C_DIS
LIN {X 0.167,Y -540.985,Z 1106.538,A 0.000,B 0.000,C 90.000,E1 312.852} C_DIS
LIN {X -0.040,Y -540.129,Z 1106.537,A 0.000,B 0.000,C 90.000,E1 312.732} C_DIS
LIN {X -0.031,Y -538.942,Z 1106.536,A 0.000,B 0.000,C 90.000,E1 312.447} C_DIS
LIN {X 0.154,Y -538.236,Z 1106.535,A 0.000,B 0.000,C 90.000,E1 312.285} C_DIS
LIN {X 0.158,Y -537.077,Z 1106.533,A 0.000,B 0.000,C 90.000,E1 312.000} C_DIS
LIN {X 0.116,Y -535.263,Z 1106.530,A 0.000,B 0.000,C 90.000,E1 311.434} C_DIS
LIN {X -0.301,Y -533.394,Z 1106.526,A 0.000,B 0.000,C 90.000,E1 310.620} C_DIS
LIN {X 0.036,Y -532.851,Z 1106.524,A 0.000,B 0.000,C 90.000,E1 310.297} C_DIS
LIN {X 0.016,Y -532.193,Z 1106.521,A 0.000,B 0.000,C 90.000,E1 309.725} C_DIS
LIN {X 0.007,Y -532.104,Z 1106.519,A 0.000,B 0.000,C 90.000,E1 309.439} C_DIS
LIN {X 0.160,Y -531.626,Z 1106.517,A 0.000,B 0.000,C 90.000,E1 308.991} C_DIS
LIN {X 0.134,Y -531.635,Z 1106.515,A 0.000,B 0.000,C 90.000,E1 308.669} C_DIS
LIN {X 0.109,Y -531.313,Z 1106.512,A 0.000,B 0.000,C 90.000,E1 308.096} C_DIS
LIN {X 0.085,Y -531.280,Z 1106.509,A 0.000,B 0.000,C 90.000,E1 307.523} C_DIS
LIN {X 0.039,Y -531.393,Z 1106.502,A 0.000,B 0.000,C 90.000,E1 306.377} C_DIS
LIN {X 0.079,Y -532.334,Z 1106.489,A 0.000,B 0.000,C 90.000,E1 304.072} C_DIS
LIN {X 0.173,Y -533.122,Z 1106.481,A 0.000,B 0.000,C 90.000,E1 302.625} C_DIS
LIN {X -0.314,Y -534.634,Z 1106.470,A 0.000,B 0.000,C 90.000,E1 300.669} C_DIS
LIN {X -0.014,Y -535.630,Z 1106.462,A 0.000,B 0.000,C 90.000,E1 299.205} C_DIS
LIN {X -0.130,Y -536.161,Z 1106.458,A 0.000,B 0.000,C 90.000,E1 298.359} C_DIS
LIN {X -0.146,Y -537.155,Z 1106.446,A 0.000,B 0.000,C 90.000,E1 296.360} C_DIS
LIN {X 0.170,Y -537.728,Z 1106.438,A 0.000,B 0.000,C 90.000,E1 294.899} C_DIS
LIN {X -0.003,Y -538.139,Z 1106.429,A 0.000,B 0.000,C 90.000,E1 293.206} C_DIS
LIN {X -0.119,Y -538.317,Z 1106.423,A 0.000,B 0.000,C 90.000,E1 292.078} C_DIS
LIN {X 0.066,Y -538.492,Z 1106.416,A 0.000,B 0.000,C 90.000,E1 290.918} C_DIS
LIN {X 0.257,Y -538.460,Z 1106.410,A 0.000,B 0.000,C 90.000,E1 289.758} C_DIS
LIN {X 0.193,Y -538.186,Z 1106.401,A 0.000,B 0.000,C 90.000,E1 288.055} C_DIS
LIN {X -0.261,Y -537.838,Z 1106.393,A 0.000,B 0.000,C 90.000,E1 286.677} C_DIS
LIN {X 0.255,Y -537.475,Z 1106.386,A 0.000,B 0.000,C 90.000,E1 285.481} C_DIS
LIN {X 0.162,Y -536.852,Z 1106.378,A 0.000,B 0.000,C 90.000,E1 284.064} C_DIS
LIN {X 0.115,Y -536.052,Z 1106.369,A 0.000,B 0.000,C 90.000,E1 282.355} C_DIS
LIN {X -0.124,Y -535.334,Z 1106.361,A 0.000,B 0.000,C 90.000,E1 280.950} C_DIS
LIN {X 0.107,Y -534.477,Z 1106.351,A 0.000,B 0.000,C 90.000,E1 279.208} C_DIS
LIN {X -0.284,Y -533.650,Z 1106.342,A 0.000,B 0.000,C 90.000,E1 277.530} C_DIS
LIN {X -0.203,Y -532.928,Z 1106.334,A 0.000,B 0.000,C 90.000,E1 276.087} C_DIS
LIN {X -0.145,Y -532.279,Z 1106.326,A 0.000,B 0.000,C 90.000,E1 274.645} C_DIS
LIN {X -0.168,Y -531.474,Z 1106.316,A 0.000,B 0.000,C 90.000,E1 272.922} C_DIS
LIN {X -0.251,Y -530.551,Z 1106.305,A 0.000,B 0.000,C 90.000,E1 270.917} C_DIS
LIN {X 0.168,Y -529.584,Z 1106.294,A 0.000,B 0.000,C 90.000,E1 268.854} C_DIS
LIN {X 0.083,Y -528.796,Z 1106.286,A 0.000,B 0.000,C 90.000,E1 267.421} C_DIS
LIN {X -0.045,Y -527.583,Z 1106.275,A 0.000,B 0.000,C 90.000,E1 265.412} C_DIS
LIN {X -0.097,Y -526.832,Z 1106.268,A 0.000,B 0.000,C 90.000,E1 264.261} C_DIS
LIN {X -0.112,Y -526.085,Z 1106.263,A 0.000,B 0.000,C 90.000,E1 263.394} C_DIS
LIN {X -0.186,Y -524.942,Z 1106.257,A 0.000,B 0.000,C 90.000,E1 262.243} C_DIS
LIN {X -0.177,Y -522.869,Z 1106.245,A 0.000,B 0.000,C 90.000,E1 260.208} C_DIS
LIN {X -0.229,Y -521.513,Z 1106.237,A 0.000,B 0.000,C 90.000,E1 258.757} C_DIS
LIN {X -0.102,Y -519.838,Z 1106.228,A 0.000,B 0.000,C 90.000,E1 256.992} C_DIS
LIN {X -0.010,Y -518.170,Z 1106.218,A 0.000,B 0.000,C 90.000,E1 255.227} C_DIS
LIN {X -0.209,Y -516.011,Z 1106.207,A 0.000,B 0.000,C 90.000,E1 253.196} C_DIS
LIN {X 0.060,Y -514.141,Z 1106.197,A 0.000,B 0.000,C 90.000,E1 251.402} C_DIS
LIN {X -0.110,Y -512.923,Z 1106.190,A 0.000,B 0.000,C 90.000,E1 250.242} C_DIS
LIN {X -0.064,Y -510.804,Z 1106.180,A 0.000,B 0.000,C 90.000,E1 248.465} C_DIS
LIN {X 0.019,Y -509.075,Z 1106.172,A 0.000,B 0.000,C 90.000,E1 246.975} C_DIS
LIN {X -0.036,Y -507.361,Z 1106.166,A 0.000,B 0.000,C 90.000,E1 245.793} C_DIS
LIN {X 0.092,Y -505.638,Z 1106.159,A 0.000,B 0.000,C 90.000,E1 244.588} C_DIS
LIN {X -0.181,Y -503.210,Z 1106.151,A 0.000,B 0.000,C 90.000,E1 243.127} C_DIS
LIN {X 0.022,Y -500.320,Z 1106.141,A 0.000,B 0.000,C 90.000,E1 241.307} C_DIS
LIN {X 0.281,Y -496.274,Z 1106.127,A 0.000,B 0.000,C 90.000,E1 238.869} C_DIS
LIN {X 0.125,Y -493.593,Z 1106.119,A 0.000,B 0.000,C 90.000,E1 237.375} C_DIS
LIN {X -0.079,Y -490.974,Z 1106.110,A 0.000,B 0.000,C 90.000,E1 235.881} C_DIS
LIN {X -0.067,Y -488.140,Z 1106.102,A 0.000,B 0.000,C 90.000,E1 234.356} C_DIS
LIN {X -0.217,Y -485.286,Z 1106.094,A 0.000,B 0.000,C 90.000,E1 232.844} C_DIS
LIN {X -0.237,Y -482.876,Z 1106.087,A 0.000,B 0.000,C 90.000,E1 231.618} C_DIS
LIN {X -0.186,Y -479.769,Z 1106.078,A 0.000,B 0.000,C 90.000,E1 230.070} C_DIS
LIN {X 0.111,Y -476.776,Z 1106.069,A 0.000,B 0.000,C 90.000,E1 228.485} C_DIS
LIN {X 0.280,Y -472.001,Z 1106.056,A 0.000,B 0.000,C 90.000,E1 225.972} C_DIS
LIN {X -0.027,Y -469.759,Z 1106.049,A 0.000,B 0.000,C 90.000,E1 224.757} C_DIS
LIN {X 0.048,Y -466.926,Z 1106.040,A 0.000,B 0.000,C 90.000,E1 223.176} C_DIS
LIN {X -0.187,Y -463.547,Z 1106.029,A 0.000,B 0.000,C 90.000,E1 221.310} C_DIS
LIN {X -0.030,Y -459.334,Z 1106.015,A 0.000,B 0.000,C 90.000,E1 218.749} C_DIS
LIN {X -0.058,Y -456.805,Z 1106.006,A 0.000,B 0.000,C 90.000,E1 217.156} C_DIS
LIN {X 0.045,Y -453.382,Z 1105.994,A 0.000,B 0.000,C 90.000,E1 214.898} C_DIS
LIN {X 0.086,Y -450.462,Z 1105.983,A 0.000,B 0.000,C 90.000,E1 212.959} C_DIS
LIN {X 0.193,Y -447.735,Z 1105.972,A 0.000,B 0.000,C 90.000,E1 211.003} C_DIS
LIN {X -0.086,Y -444.392,Z 1105.958,A 0.000,B 0.000,C 90.000,E1 208.437} C_DIS
LIN {X -0.023,Y -442.610,Z 1105.949,A 0.000,B 0.000,C 90.000,E1 206.796} C_DIS
LIN {X 0.000,Y -441.109,Z 1105.940,A 0.000,B 0.000,C 90.000,E1 205.155} C_DIS
LIN {X 0.154,Y -440.429,Z 1105.932,A 0.000,B 0.000,C 90.000,E1 203.823} C_DIS
LIN {X -0.036,Y -440.657,Z 1105.923,A 0.000,B 0.000,C 90.000,E1 202.206} C_DIS
LIN {X -0.232,Y -441.806,Z 1105.916,A 0.000,B 0.000,C 90.000,E1 200.918} C_DIS
LIN {X 0.154,Y -443.538,Z 1105.911,A 0.000,B 0.000,C 90.000,E1 199.885} C_DIS
LIN {X 0.144,Y -445.836,Z 1105.905,A 0.000,B 0.000,C 90.000,E1 198.906} C_DIS
LIN {X 0.016,Y -448.628,Z 1105.900,A 0.000,B 0.000,C 90.000,E1 197.946} C_DIS
LIN {X -0.138,Y -455.304,Z 1105.889,A 0.000,B 0.000,C 90.000,E1 196.024} C_DIS
LIN {X -0.113,Y -465.442,Z 1105.875,A 0.000,B 0.000,C 90.000,E1 193.467} C_DIS
LIN {X 0.055,Y -479.054,Z 1105.857,A 0.000,B 0.000,C 90.000,E1 190.310} C_DIS
LIN {X -0.126,Y -484.643,Z 1105.850,A 0.000,B 0.000,C 90.000,E1 189.095} C_DIS
LIN {X 0.000,Y -490.930,Z 1105.843,A 0.000,B 0.000,C 90.000,E1 187.701} C_DIS
LIN {X 0.162,Y -497.112,Z 1105.835,A 0.000,B 0.000,C 90.000,E1 186.315} C_DIS
LIN {X -0.010,Y -505.057,Z 1105.825,A 0.000,B 0.000,C 90.000,E1 184.531} C_DIS
LIN {X 0.252,Y -512.432,Z 1105.816,A 0.000,B 0.000,C 90.000,E1 182.865} C_DIS
LIN {X 0.068,Y -521.051,Z 1105.806,A 0.000,B 0.000,C 90.000,E1 180.974} C_DIS
LIN {X 0.139,Y -527.112,Z 1105.798,A 0.000,B 0.000,C 90.000,E1 179.656} C_DIS
LIN {X 0.034,Y -533.763,Z 1105.790,A 0.000,B 0.000,C 90.000,E1 178.224} C_DIS
LIN {X -0.215,Y -539.726,Z 1105.783,A 0.000,B 0.000,C 90.000,E1 176.963} C_DIS
LIN {X 0.209,Y -545.643,Z 1105.776,A 0.000,B 0.000,C 90.000,E1 175.641} C_DIS
LIN {X 0.048,Y -553.399,Z 1105.767,A 0.000,B 0.000,C 90.000,E1 173.970} C_DIS
LIN {X 0.294,Y -560.568,Z 1105.758,A 0.000,B 0.000,C 90.000,E1 172.413} C_DIS
LIN {X -0.133,Y -565.088,Z 1105.753,A 0.000,B 0.000,C 90.000,E1 171.489} C_DIS
LIN {X 0.084,Y -571.341,Z 1105.745,A 0.000,B 0.000,C 90.000,E1 170.095} C_DIS
LIN {X 0.290,Y -578.096,Z 1105.737,A 0.000,B 0.000,C 90.000,E1 168.578} C_DIS
LIN {X 0.047,Y -582.789,Z 1105.731,A 0.000,B 0.000,C 90.000,E1 167.521} C_DIS
LIN {X 0.188,Y -586.208,Z 1105.726,A 0.000,B 0.000,C 90.000,E1 166.700} C_DIS
LIN {X 0.044,Y -590.546,Z 1105.720,A 0.000,B 0.000,C 90.000,E1 165.644} C_DIS
LIN {X 0.104,Y -594.684,Z 1105.714,A 0.000,B 0.000,C 90.000,E1 164.574} C_DIS
LIN {X 0.222,Y -598.607,Z 1105.708,A 0.000,B 0.000,C 90.000,E1 163.504} C_DIS
LIN {X 0.100,Y -601.355,Z 1105.704,A 0.000,B 0.000,C 90.000,E1 162.725} C_DIS
LIN {X -0.086,Y -604.868,Z 1105.698,A 0.000,B 0.000,C 90.000,E1 161.692} C_DIS
LIN {X 0.084,Y -608.910,Z 1105.691,A 0.000,B 0.000,C 90.000,E1 160.369} C_DIS
LIN {X -0.001,Y -611.995,Z 1105.685,A 0.000,B 0.000,C 90.000,E1 159.337} C_DIS
LIN {X 0.174,Y -614.927,Z 1105.679,A 0.000,B 0.000,C 90.000,E1 158.284} C_DIS
LIN {X 0.133,Y -618.458,Z 1105.672,A 0.000,B 0.000,C 90.000,E1 156.997} C_DIS
LIN {X -0.183,Y -621.865,Z 1105.665,A 0.000,B 0.000,C 90.000,E1 155.741} C_DIS
LIN {X -0.177,Y -625.118,Z 1105.658,A 0.000,B 0.000,C 90.000,E1 154.460} C_DIS
LIN {X -0.122,Y -627.662,Z 1105.652,A 0.000,B 0.000,C 90.000,E1 153.435} C_DIS
LIN {X -0.059,Y -629.428,Z 1105.648,A 0.000,B 0.000,C 90.000,E1 152.666} C_DIS
LIN {X 0.110,Y -632.818,Z 1105.640,A 0.000,B 0.000,C 90.000,E1 151.129} C_DIS
LIN {X 0.046,Y -635.609,Z 1105.633,A 0.000,B 0.000,C 90.000,E1 149.871} C_DIS
LIN {X 0.028,Y -638.213,Z 1105.626,A 0.000,B 0.000,C 90.000,E1 148.614} C_DIS
LIN {X -0.155,Y -640.711,Z 1105.619,A 0.000,B 0.000,C 90.000,E1 147.375} C_DIS
LIN {X -0.239,Y -643.599,Z 1105.610,A 0.000,B 0.000,C 90.000,E1 145.881} C_DIS
LIN {X 0.146,Y -645.388,Z 1105.605,A 0.000,B 0.000,C 90.000,E1 144.848} C_DIS
LIN {X 0.358,Y -648.058,Z 1105.597,A 0.000,B 0.000,C 90.000,E1 143.336} C_DIS
LIN {X -0.279,Y -650.696,Z 1105.588,A 0.000,B 0.000,C 90.000,E1 141.904} C_DIS
LIN {X -0.023,Y -653.924,Z 1105.579,A 0.000,B 0.000,C 90.000,E1 140.150} C_DIS
LIN {X 0.224,Y -657.242,Z 1105.569,A 0.000,B 0.000,C 90.000,E1 138.405} C_DIS
LIN {X 0.057,Y -660.685,Z 1105.560,A 0.000,B 0.000,C 90.000,E1 136.701} C_DIS
LIN {X -0.065,Y -665.470,Z 1105.547,A 0.000,B 0.000,C 90.000,E1 134.514} C_DIS
LIN {X 0.429,Y -670.089,Z 1105.536,A 0.000,B 0.000,C 90.000,E1 132.528} C_DIS
LIN {X 0.121,Y -674.318,Z 1105.527,A 0.000,B 0.000,C 90.000,E1 130.862} C_DIS
LIN {X -0.115,Y -677.867,Z 1105.519,A 0.000,B 0.000,C 90.000,E1 129.439} C_DIS
LIN {X 0.270,Y -682.202,Z 1105.510,A 0.000,B 0.000,C 90.000,E1 127.729} C_DIS
LIN {X -0.291,Y -685.267,Z 1105.503,A 0.000,B 0.000,C 90.000,E1 126.583} C_DIS
LIN {X 0.341,Y -688.835,Z 1105.495,A 0.000,B 0.000,C 90.000,E1 125.105} C_DIS
LIN {X 0.081,Y -692.268,Z 1105.487,A 0.000,B 0.000,C 90.000,E1 123.706} C_DIS
LIN {X 0.082,Y -695.723,Z 1105.479,A 0.000,B 0.000,C 90.000,E1 122.291} C_DIS
LIN {X 0.247,Y -697.935,Z 1105.474,A 0.000,B 0.000,C 90.000,E1 121.337} C_DIS
LIN {X 0.076,Y -699.772,Z 1105.469,A 0.000,B 0.000,C 90.000,E1 120.413} C_DIS
LIN {X -0.069,Y -701.400,Z 1105.464,A 0.000,B 0.000,C 90.000,E1 119.489} C_DIS
LIN {X -0.195,Y -702.835,Z 1105.459,A 0.000,B 0.000,C 90.000,E1 118.565} C_DIS
LIN {X -0.311,Y -704.009,Z 1105.453,A 0.000,B 0.000,C 90.000,E1 117.641} C_DIS
LIN {X -0.083,Y -704.674,Z 1105.450,A 0.000,B 0.000,C 90.000,E1 116.924} C_DIS
LIN {X 0.412,Y -705.517,Z 1105.443,A 0.000,B 0.000,C 90.000,E1 115.720} C_DIS
LIN {X 0.342,Y -705.793,Z 1105.439,A 0.000,B 0.000,C 90.000,E1 115.027} C_DIS
LIN {X -0.012,Y -705.735,Z 1105.437,A 0.000,B 0.000,C 90.000,E1 114.591} C_DIS
LIN {X -0.077,Y -705.047,Z 1105.434,A 0.000,B 0.000,C 90.000,E1 114.131} C_DIS
LIN {X -0.077,Y -704.546,Z 1105.433,A 0.000,B 0.000,C 90.000,E1 113.898} C_DIS
LIN {X -0.153,Y -702.723,Z 1105.430,A 0.000,B 0.000,C 90.000,E1 113.439} C_DIS
LIN {X -0.293,Y -702.178,Z 1105.430,A 0.000,B 0.000,C 90.000,E1 113.334} C_DIS
LIN {X -0.153,Y -701.340,Z 1105.429,A 0.000,B 0.000,C 90.000,E1 113.206} C_DIS
LIN {X 0.114,Y -697.203,Z 1105.426,A 0.000,B 0.000,C 90.000,E1 112.717} C_DIS
LIN {X 0.242,Y -695.709,Z 1105.426,A 0.000,B 0.000,C 90.000,E1 112.589} C_DIS
LIN {X -0.271,Y -693.232,Z 1105.425,A 0.000,B 0.000,C 90.000,E1 112.514} C_DIS
LIN {X 0.003,Y -686.151,Z 1105.423,A 0.000,B 0.000,C 90.000,E1 112.206} C_DIS
LIN {X 0.008,Y -683.653,Z 1105.423,A 0.000,B 0.000,C 90.000,E1 112.153} C_DIS
LIN {X -0.096,Y -676.270,Z 1105.423,A 0.000,B 0.000,C 90.000,E1 112.078} C_DIS
LIN {X -0.136,Y -604.109,Z 1105.423,A 0.000,B 0.000,C 90.000,E1 112.078} C_DIS
LIN {X 0.179,Y -600.395,Z 1105.422,A 0.000,B 0.000,C 90.000,E1 111.844} C_DIS
LIN {X 0.106,Y -595.944,Z 1105.420,A 0.000,B 0.000,C 90.000,E1 111.535} C_DIS
LIN {X -0.294,Y -578.340,Z 1105.411,A 0.000,B 0.000,C 90.000,E1 110.066} C_DIS
LIN {X -0.050,Y -574.052,Z 1105.409,A 0.000,B 0.000,C 90.000,E1 109.685} C_DIS
LIN {X 0.177,Y -567.992,Z 1105.407,A 0.000,B 0.000,C 90.000,E1 109.214} C_DIS
LIN {X -0.114,Y -561.512,Z 1105.405,A 0.000,B 0.000,C 90.000,E1 108.833} C_DIS
LIN {X 0.231,Y -554.779,Z 1105.402,A 0.000,B 0.000,C 90.000,E1 108.417} C_DIS
LIN {X -0.165,Y -549.997,Z 1105.401,A 0.000,B 0.000,C 90.000,E1 108.109} C_DIS
LIN {X 0.153,Y -548.580,Z 1105.399,A 0.000,B 0.000,C 90.000,E1 107.873} C_DIS
LIN {X 0.111,Y -548.560,Z 1105.399,A 0.000,B 0.000,C 90.000,E1 107.873} C_DIS
LIN {X -0.220,Y -548.218,Z 1105.398,A 0.000,B 0.000,C 90.000,E1 107.583} C_DIS
LIN {X 0.079,Y -548.646,Z 1105.392,A 0.000,B 0.000,C 90.000,E1 106.567} C_DIS
LIN {X 0.161,Y -550.031,Z 1105.381,A 0.000,B 0.000,C 90.000,E1 104.592} C_DIS
LIN {X -0.013,Y -551.560,Z 1105.370,A 0.000,B 0.000,C 90.000,E1 102.647} C_DIS
LIN {X 0.272,Y -553.374,Z 1105.359,A 0.000,B 0.000,C 90.000,E1 100.658} C_DIS
LIN {X -0.008,Y -555.652,Z 1105.347,A 0.000,B 0.000,C 90.000,E1 98.454} C_DIS
LIN {X 0.189,Y -557.684,Z 1105.336,A 0.000,B 0.000,C 90.000,E1 96.486} C_DIS
LIN {X 0.101,Y -559.035,Z 1105.328,A 0.000,B 0.000,C 90.000,E1 95.106} C_DIS
LIN {X 0.039,Y -560.168,Z 1105.321,A 0.000,B 0.000,C 90.000,E1 93.726} C_DIS
LIN {X -0.131,Y -560.906,Z 1105.315,A 0.000,B 0.000,C 90.000,E1 92.636} C_DIS
LIN {X 0.172,Y -561.415,Z 1105.310,A 0.000,B 0.000,C 90.000,E1 91.776} C_DIS
LIN {X 0.200,Y -562.338,Z 1105.301,A 0.000,B 0.000,C 90.000,E1 90.115} C_DIS
LIN {X 0.248,Y -563.091,Z 1105.292,A 0.000,B 0.000,C 90.000,E1 88.453} C_DIS
LIN {X 0.219,Y -563.764,Z 1105.284,A 0.000,B 0.000,C 90.000,E1 87.078} C_DIS
LIN {X -0.080,Y -564.590,Z 1105.273,A 0.000,B 0.000,C 90.000,E1 85.179} C_DIS
LIN {X -0.042,Y -565.140,Z 1105.266,A 0.000,B 0.000,C 90.000,E1 83.799} C_DIS
LIN {X -0.244,Y -565.814,Z 1105.255,A 0.000,B 0.000,C 90.000,E1 81.894} C_DIS
LIN {X -0.046,Y -566.260,Z 1105.247,A 0.000,B 0.000,C 90.000,E1 80.500} C_DIS
LIN {X -0.046,Y -567.114,Z 1105.237,A 0.000,B 0.000,C 90.000,E1 78.578} C_DIS
LIN {X 0.258,Y -568.207,Z 1105.224,A 0.000,B 0.000,C 90.000,E1 76.353} C_DIS
LIN {X -0.242,Y -569.425,Z 1105.212,A 0.000,B 0.000,C 90.000,E1 74.212} C_DIS
LIN {X 0.005,Y -571.075,Z 1105.200,A 0.000,B 0.000,C 90.000,E1 72.000} C_DIS
LIN {X 0.313,Y -572.152,Z 1105.193,A 0.000,B 0.000,C 90.000,E1 70.604} C_DIS
LIN {X 0.089,Y -573.878,Z 1105.182,A 0.000,B 0.000,C 90.000,E1 68.720} C_DIS
LIN {X -0.051,Y -575.304,Z 1105.173,A 0.000,B 0.000,C 90.000,E1 67.102} C_DIS
LIN {X 0.147,Y -576.200,Z 1105.167,A 0.000,B 0.000,C 90.000,E1 65.997} C_DIS
LIN {X -0.089,Y -577.315,Z 1105.159,A 0.000,B 0.000,C 90.000,E1 64.665} C_DIS
LIN {X -0.190,Y -578.495,Z 1105.150,A 0.000,B 0.000,C 90.000,E1 63.050} C_DIS
LIN {X -0.117,Y -579.464,Z 1105.143,A 0.000,B 0.000,C 90.000,E1 61.691} C_DIS
LIN {X -0.178,Y -580.471,Z 1105.134,A 0.000,B 0.000,C 90.000,E1 60.078} C_DIS
LIN {X -0.303,Y -581.248,Z 1105.126,A 0.000,B 0.000,C 90.000,E1 58.742} C_DIS
LIN {X -0.271,Y -581.868,Z 1105.120,A 0.000,B 0.000,C 90.000,E1 57.661} C_DIS
LIN {X 0.132,Y -582.964,Z 1105.108,A 0.000,B 0.000,C 90.000,E1 55.468} C_DIS
LIN {X -0.240,Y -583.805,Z 1105.098,A 0.000,B 0.000,C 90.000,E1 53.623} C_DIS
LIN {X 0.038,Y -584.362,Z 1105.089,A 0.000,B 0.000,C 90.000,E1 51.984} C_DIS
LIN {X 0.130,Y -584.550,Z 1105.084,A 0.000,B 0.000,C 90.000,E1 51.170} C_DIS
LIN {X -0.042,Y -584.550,Z 1105.078,A 0.000,B 0.000,C 90.000,E1 50.114} C_DIS
LIN {X 0.233,Y -584.427,Z 1105.073,A 0.000,B 0.000,C 90.000,E1 49.013} C_DIS
LIN {X -0.207,Y -584.139,Z 1105.065,A 0.000,B 0.000,C 90.000,E1 47.715} C_DIS
LIN {X -0.260,Y -583.687,Z 1105.058,A 0.000,B 0.000,C 90.000,E1 46.377} C_DIS
LIN {X 0.087,Y -582.978,Z 1105.050,A 0.000,B 0.000,C 90.000,E1 45.000} C_DIS
LIN {X -0.138,Y -582.257,Z 1105.044,A 0.000,B 0.000,C 90.000,E1 43.947} C_DIS
LIN {X 0.045,Y -581.177,Z 1105.038,A 0.000,B 0.000,C 90.000,E1 42.852} C_DIS
LIN {X 0.055,Y -580.287,Z 1105.034,A 0.000,B 0.000,C 90.000,E1 42.043} C_DIS
LIN {X -0.181,Y -578.894,Z 1105.028,A 0.000,B 0.000,C 90.000,E1 40.987} C_DIS
LIN {X -0.148,Y -577.752,Z 1105.023,A 0.000,B 0.000,C 90.000,E1 40.172} C_DIS
LIN {X -0.263,Y -575.442,Z 1105.016,A 0.000,B 0.000,C 90.000,E1 38.830} C_DIS
LIN {X 0.025,Y -572.619,Z 1105.008,A 0.000,B 0.000,C 90.000,E1 37.443} C_DIS
LIN {X -0.015,Y -570.575,Z 1105.004,A 0.000,B 0.000,C 90.000,E1 36.629} C_DIS
LIN {X -0.087,Y -569.097,Z 1105.000,A 0.000,B 0.000,C 90.000,E1 36.091} C_DIS
LIN {X 0.168,Y -567.409,Z 1104.997,A 0.000,B 0.000,C 90.000,E1 35.518} C_DIS
LIN {X 0.310,Y -563.516,Z 1104.991,A 0.000,B 0.000,C 90.000,E1 34.405} C_DIS
LIN {X -0.365,Y -562.514,Z 1104.990,A 0.000,B 0.000,C 90.000,E1 34.199} C_DIS
LIN {X -0.164,Y -560.241,Z 1104.987,A 0.000,B 0.000,C 90.000,E1 33.627} C_DIS
LIN {X 0.259,Y -556.511,Z 1104.982,A 0.000,B 0.000,C 90.000,E1 32.752} C_DIS
LIN {X -0.012,Y -553.215,Z 1104.978,A 0.000,B 0.000,C 90.000,E1 32.084} C_DIS
LIN {X -0.138,Y -548.913,Z 1104.974,A 0.000,B 0.000,C 90.000,E1 31.258} C_DIS
LIN {X 0.001,Y -545.051,Z 1104.970,A 0.000,B 0.000,C 90.000,E1 30.541} C_DIS
LIN {X 0.113,Y -539.339,Z 1104.964,A 0.000,B 0.000,C 90.000,E1 29.539} C_DIS
LIN {X 0.167,Y -534.828,Z 1104.960,A 0.000,B 0.000,C 90.000,E1 28.821} C_DIS
LIN {X 0.178,Y -529.914,Z 1104.956,A 0.000,B 0.000,C 90.000,E1 28.103} C_DIS
LIN {X -0.261,Y -526.757,Z 1104.954,A 0.000,B 0.000,C 90.000,E1 27.719} C_DIS
LIN {X 0.151,Y -521.161,Z 1104.950,A 0.000,B 0.000,C 90.000,E1 26.950} C_DIS
LIN {X 0.038,Y -515.072,Z 1104.946,A 0.000,B 0.000,C 90.000,E1 26.232} C_DIS
LIN {X -0.071,Y -508.548,Z 1104.942,A 0.000,B 0.000,C 90.000,E1 25.515} C_DIS
LIN {X -0.048,Y -499.079,Z 1104.936,A 0.000,B 0.000,C 90.000,E1 24.515} C_DIS
LIN {X 0.053,Y -494.931,Z 1104.934,A 0.000,B 0.000,C 90.000,E1 24.079} C_DIS
LIN {X 0.027,Y -486.436,Z 1104.929,A 0.000,B 0.000,C 90.000,E1 23.259} C_DIS
LIN {X 0.160,Y -478.072,Z 1104.925,A 0.000,B 0.000,C 90.000,E1 22.461} C_DIS
LIN {X 0.266,Y -464.741,Z 1104.918,A 0.000,B 0.000,C 90.000,E1 21.280} C_DIS
LIN {X 0.208,Y -450.102,Z 1104.911,A 0.000,B 0.000,C 90.000,E1 19.993} C_DIS
LIN {X 0.005,Y -431.197,Z 1104.901,A 0.000,B 0.000,C 90.000,E1 18.236} C_DIS
LIN {X -0.050,Y -418.616,Z 1104.894,A 0.000,B 0.000,C 90.000,E1 16.913} C_DIS
LIN {X 0.057,Y -409.128,Z 1104.888,A 0.000,B 0.000,C 90.000,E1 15.788} C_DIS
LIN {X 0.136,Y -400.074,Z 1104.881,A 0.000,B 0.000,C 90.000,E1 14.592} C_DIS
LIN {X 0.119,Y -397.722,Z 1104.879,A 0.000,B 0.000,C 90.000,E1 14.245} C_DIS
LIN {X -0.150,Y -395.256,Z 1104.877,A 0.000,B 0.000,C 90.000,E1 13.828} C_DIS
LIN {X -0.073,Y -393.020,Z 1104.874,A 0.000,B 0.000,C 90.000,E1 13.244} C_DIS
LIN {X -0.006,Y -392.156,Z 1104.871,A 0.000,B 0.000,C 90.000,E1 12.703} C_DIS
LIN {X -0.036,Y -392.037,Z 1104.868,A 0.000,B 0.000,C 90.000,E1 12.175} C_DIS
LIN {X -0.115,Y -392.355,Z 1104.865,A 0.000,B 0.000,C 90.000,E1 11.771} C_DIS
LIN {X -0.206,Y -393.289,Z 1104.861,A 0.000,B 0.000,C 90.000,E1 11.074} C_DIS
LIN {X 0.035,Y -397.331,Z 1104.850,A 0.000,B 0.000,C 90.000,E1 8.916} C_DIS
LIN {X -0.141,Y -402.388,Z 1104.838,A 0.000,B 0.000,C 90.000,E1 6.834} C_DIS
LIN {X 0.194,Y -404.895,Z 1104.832,A 0.000,B 0.000,C 90.000,E1 5.739} C_DIS
LIN {X 0.171,Y -406.405,Z 1104.829,A 0.000,B 0.000,C 90.000,E1 5.220} C_DIS
LIN {X -0.196,Y -408.014,Z 1104.827,A 0.000,B 0.000,C 90.000,E1 4.878} C_DIS
LIN {X -0.190,Y -409.737,Z 1104.825,A 0.000,B 0.000,C 90.000,E1 4.531} C_DIS
LIN {X -0.209,Y -412.044,Z 1104.823,A 0.000,B 0.000,C 90.000,E1 4.188} C_DIS
LIN {X 0.027,Y -417.353,Z 1104.820,A 0.000,B 0.000,C 90.000,E1 3.669} C_DIS
LIN {X -0.163,Y -425.905,Z 1104.817,A 0.000,B 0.000,C 90.000,E1 3.094} C_DIS
LIN {X 0.183,Y -445.649,Z 1104.810,A 0.000,B 0.000,C 90.000,E1 1.718} C_DIS
LIN {X 0.021,Y -463.716,Z 1104.803,A 0.000,B 0.000,C 90.000,E1 0.573} C_DIS
LIN {X -0.083,Y -479.288,Z 1104.798,A 0.000,B 0.000,C 90.000,E1 359.599} C_DIS
